# B&R Automation Studio project Genmot_Markalama_
Automation Studio 3.0.90.36 SP18

## Configuration Config1

### Task classes (Cpu.sw)
```
Cyclic#1:
  PowerAx1 <- PowerAx1.prg
  PowerAx2 <- PowerAx2.prg
  RZAxisCont <- RZAxisControl.prg
  RYAxisCont <- RYAxisControl.prg
  RXAxisCont <- RXAxisControl.prg
  RAAxisCont <- RAAxisControl.prg
  RC1AxisCon <- RC1AxisControl.prg
  RC2AxisCon <- RC2AxisControl.prg
  GRXAxisCon <- GRXAxisControl.prg
  GRZAxisCon <- GRZAxisControl.prg
  Master <- Master.prg
Cyclic#2:
  Sender <- LibDVFrame1_ST.Sender.prg
  Receiver <- LibDVFrame1_ST.Receiver.prg
Cyclic#4:
  GRYAxisCon <- GRYAxisControl.prg
DataObjects: Acp10sys
NcDataObjects: acp10etxen <- acp10etxen.dob, gaxis01i <- RYAxisobj.gaxis01i.dob, gaxis01a <- RYAxisobj.gaxis01a.dob, gaxis02i <- RAAxisobj.gaxis02i.dob, gaxis02a <- RAAxisobj.gaxis02a.dob, gaxis03i <- RXAxisobj.gaxis03i.dob, gaxis03a <- RXAxisobj.gaxis03a.dob, gz1_axisi <- RZAxisobj.gz1_axisi.dob, gz1_axisa <- RZAxisobj.gz1_axisa.dob, gc1_axisi <- RC1Axisobj.gc1_axisi.dob, gc2_axisa <- RC1Axisobj.gc2_axisa.dob, gc2_axisi <- RC2Axisobj.gc2_axisi.dob, gc2_axisa1 <- RC2Axisobj.gc2_axisa.dob, powersp1i <- PowerSp1obj.powersp1i.dob, powersp1a <- PowerSp1obj.powersp1a.dob, powersp2i <- PowerSp2obj.powersp2i.dob, powersp2a <- PowerSp2obj.powersp2a.dob, grx_axisi <- GRXAxisobj.grx_axisi.dob, grx_axisa <- GRXAxisobj.grx_axisa.dob, grz_axisi <- GRZAxisobj.grz_axisi.dob, grz_axisa <- GRZAxisobj.grz_axisa.dob, gry_axisi <- GRYAxisobj.gry_axisi.dob, gry_axisa <- GRYAxisobj.gry_axisa.dob
Binaries: AsOPCC, ashwd, arconfig, sysconf, asfw, iomap, Acp10cfg, Acp10map, Visu03, vcctrend, vccline, vcchtml, vcbclass, vccbmp, vcclbox, vccalarm, vcrt, vcshared, vcnet, arialbd, vcdsloc, vcgclass, vcresman, vccstr, vcmgr, vcfile, vcalarm, vccurl, vcpdsw, Visu02, vcpdvnc, vcdsint, vccnum, vccbtn, vcpfar10, vcpkat, vctcal, arial, vccovl, vcctext, vccshape, vcfntttf, vcxml, Visu01, visvc, vccbar
Libraries: acp10_mc, brsystem, Acp10man, sys_lib, NcGlobal, Acp10par, runtime, Acp10sdc, standard, asstring, astime, powerlnk, AsWeigh, AsBrMath, LoopConR, AsBrStr, FileIO, AsEPL, AsARCfg, asieccon, dvframe, ashw, dataobj, visapi
```

### Cpu.per - PLC1/Cpu.per
```iecst
(********************************************************************
 * COPYRIGHT --
 ********************************************************************
 * File: Cpu.per
 * Author: Coder
 * Created: September 22, 2013
 ********************************************************************
 * Declaration of permanent variables
 ********************************************************************)
VAR_CONFIG
	Retain AT %M0;
	Eksen_Hizlari AT %M76;
END_VAR
```

### IoMap.iom - PLC1/IoMap.iom
```iecst
(********************************************************************
 * COPYRIGHT --
 ********************************************************************
 * File: IoMap.iom
 * Author: Coder
 * Created: September 22, 2013
 ********************************************************************
 * IO mapping file
 ********************************************************************)
VAR_CONFIG
	DI.Acil_Stop AT %IX.SL1.IF1.ST1.IF1.ST2.DigitalInput01;
	DI.X_PosLimit AT %IX.SL1.IF1.ST1.IF1.ST2.DigitalInput03;
	DI.X_NegLimit AT %IX.SL1.IF1.ST1.IF1.ST2.DigitalInput04;
	DI.X_RefSensor AT %IX.SL1.IF1.ST1.IF1.ST2.DigitalInput02;
	DI.Y_NegLimit AT %IX.SL1.IF1.ST1.IF1.ST2.DigitalInput06;
	DI.Y_RefSensor AT %IX.SL1.IF1.ST1.IF1.ST2.DigitalInput05;
	DI.Y_PosLimit AT %IX.SL1.IF1.ST1.IF1.ST2.DigitalInput07;
	DI.Lazer_IsBitti AT %IX.SL1.IF1.ST1.IF1.ST2.DigitalInput08;
	DI.GRX_PosLimit AT %IX.SL1.IF1.ST1.IF1.ST3.DigitalInput01;
	DI.GRX_RefSensor AT %IX.SL1.IF1.ST1.IF1.ST2.DigitalInput12;
	DI.GRX_NegLimit AT %IX.SL1.IF1.ST1.IF1.ST2.DigitalInput11;
	DI.GRZ_PosLimit AT %IX.SL1.IF1.ST1.IF1.ST3.DigitalInput04;
	DI.GRZ_NegLimit AT %IX.SL1.IF1.ST1.IF1.ST3.DigitalInput03;
	DI.GRZ_RefSensor AT %IX.SL1.IF1.ST1.IF1.ST3.DigitalInput02;
	DI.GRY_NegLimit AT %IX.SL1.IF1.ST1.IF1.ST3.DigitalInput06;
	DQ.Konveyor_Ileri AT %QX.SL1.IF1.ST1.IF1.ST7.DigitalOutput01;
	DQ.Konveyor_Geri AT %QX.SL1.IF1.ST1.IF1.ST7.DigitalOutput02;
	DQ.Lazer_Start AT %QX.SL1.IF1.ST1.IF1.ST6.DigitalOutput01;
	DQ.Lazer_Stop AT %QX.SL1.IF1.ST1.IF1.ST6.DigitalOutput02;
	DQ.Lazer_Pointer AT %QX.SL1.IF1.ST1.IF1.ST6.DigitalOutput03;
	DQ.Lazer_Hatch AT %QX.SL1.IF1.ST1.IF1.ST6.DigitalOutput04;
	DQ.Lazer_Barcode AT %QX.SL1.IF1.ST1.IF1.ST6.DigitalOutput05;
	DQ.Kripper_Ac AT %QX.SL1.IF1.ST1.IF1.ST6.DigitalOutput07;
	DQ.Kripper_Kapat AT %QX.SL1.IF1.ST1.IF1.ST6.DigitalOutput08;
	DI.LAnahtarKonumu1 AT %IX.SL1.IF1.ST1.IF1.ST4.DigitalInput09;
	DI.LAnahtarKonumu2 AT %IX.SL1.IF1.ST1.IF1.ST4.DigitalInput11;
	DI.LAnahtarKonumu3 AT %IX.SL1.IF1.ST1.IF1.ST4.DigitalInput02;
	DI.LAnahtarKonumu4 AT %IX.SL1.IF1.ST1.IF1.ST4.DigitalInput04;
	DI.L_JoySag AT %IX.SL1.IF1.ST1.IF1.ST4.DigitalInput05;
	DI.L_JoySol AT %IX.SL1.IF1.ST1.IF1.ST4.DigitalInput07;
	DI.L_Input1 AT %IX.SL1.IF1.ST1.IF1.ST4.DigitalInput03;
	DI.RAnahtarKonumu1 AT %IX.SL1.IF1.ST1.IF1.ST5.DigitalInput09;
	DI.RAnahtarKonumu2 AT %IX.SL1.IF1.ST1.IF1.ST5.DigitalInput11;
	DI.RAnahtarKonumu3 AT %IX.SL1.IF1.ST1.IF1.ST5.DigitalInput02;
	DI.RAnahtarKonumu4 AT %IX.SL1.IF1.ST1.IF1.ST5.DigitalInput04;
	DI.R_JoySag AT %IX.SL1.IF1.ST1.IF1.ST5.DigitalInput05;
	DI.R_JoySol AT %IX.SL1.IF1.ST1.IF1.ST5.DigitalInput07;
	DI.R_Input1 AT %IX.SL1.IF1.ST1.IF1.ST5.DigitalInput03;
END_VAR
```

### LazerOpcMap.opcm - PLC1/LazerOpcMap.opcm
```
Map:
  CommunicationPath:
    Pvi (CommunicationTimeout=0, ProcessTimeout=0, RemoutePvi=false, IpAddress=127.0.0.1, PortNumber=20000, Others=)
    Linie LNINA2 (Type=LNINA2, CFG=, Others=)
    Device TCPIP (Type=Tcpip, IF=tcpip, BD=57600, RS=232, PA=1, CNO=0, IT=40, BI=1598, MDA=32, SA=54, CMODE=11, CT=20, MC=15, LOPO=11159, MO='Modem description see Control Panel', TN='+90909090909', MR=INFINITE, RI=60, FF=nw_load.bin, FC=nw_pb_32.br, CB=2, RC=3, TE=3000, TQ=3000, SR=0, RETRY=3, DA=2, TO=100, BA=851968, Others=)
    Station (CN=Station, MODE=SPS, DAIP=, PN=502, Others=)
    Cpu NewTCPIPConnection (CN=, SP=, RT=1000, DA=, DAIP=192.168.137.2, RW=0, REPO=11159, CKDA=1, Others=)
  Tag GC1_MoveAbsolute (Scope=)
    PVI GC1Axis.Command.MoveAbsolute (Path=GC1Axis.Command.MoveAbsolute, Type=Pvar, AccessType=DATA)
      ObjectDescriptor (VT=boolean, VN=1, VL=1, CD=GC1Axis.Command.MoveAbsolute, AT=rw, RF=1000, DV=, WR=true)
      LinkDescriptor (BitNumber=none, LT=raw)
        CastMode (Pg2000=false, Decimal=false, Range=false, Rounding=false, TerminateStrings=false)
  Tag GC1_Position (Scope=)
    PVI GC1Axis.Parameter.Position (Path=GC1Axis.Parameter.Position, Type=Pvar, AccessType=DATA)
      ObjectDescriptor (VT=f32, VN=1, VL=4, CD=GC1Axis.Parameter.Position, AT=rw, RF=1000, DV=, WR=true)
      LinkDescriptor (BitNumber=none, LT=raw)
        CastMode (Pg2000=false, Decimal=false, Range=false, Rounding=false, TerminateStrings=false)
  Tag Markalama_Ok_Delphi (Scope=)
    PVI Parametreler_0.Markalama_Ok_Delphi (Path=Parametreler_0.Markalama_Ok_Delphi, Type=Pvar, AccessType=DATA)
      ObjectDescriptor (VT=boolean, VN=1, VL=1, CD=Parametreler_0.Markalama_Ok_Delphi, AT=rw, RF=1000, DV=, WR=true)
      LinkDescriptor (BitNumber=none, LT=raw)
        CastMode (Pg2000=false, Decimal=false, Range=false, Rounding=false, TerminateStrings=false)
  Tag A_JogVelocity (Scope=)
    PVI Eksen_Hizlari.A_JogVelocity (Path=Eksen_Hizlari.A_JogVelocity, Type=Pvar, AccessType=DATA)
      ObjectDescriptor (VT=f32, VN=1, VL=4, CD=Eksen_Hizlari.A_JogVelocity, AT=rw, RF=1000, DV=, WR=true)
      LinkDescriptor (BitNumber=none, LT=raw)
        CastMode (Pg2000=false, Decimal=false, Range=false, Rounding=false, TerminateStrings=false)
  Tag A_PosVelocity (Scope=)
    PVI Eksen_Hizlari.A_PosVelocity (Path=Eksen_Hizlari.A_PosVelocity, Type=Pvar, AccessType=DATA)
      ObjectDescriptor (VT=f32, VN=1, VL=4, CD=Eksen_Hizlari.A_PosVelocity, AT=rw, RF=1000, DV=, WR=true)
      LinkDescriptor (BitNumber=none, LT=raw)
        CastMode (Pg2000=false, Decimal=false, Range=false, Rounding=false, TerminateStrings=false)
  Tag GC1_JogVelocity (Scope=)
    PVI Eksen_Hizlari.GC1_JogVelocity (Path=Eksen_Hizlari.GC1_JogVelocity, Type=Pvar, AccessType=DATA)
      ObjectDescriptor (VT=f32, VN=1, VL=4, CD=Eksen_Hizlari.GC1_JogVelocity, AT=rw, RF=1000, DV=, WR=true)
      LinkDescriptor (BitNumber=none, LT=raw)
        CastMode (Pg2000=false, Decimal=false, Range=false, Rounding=false, TerminateStrings=false)
  Tag GC1_PosVelocity (Scope=)
    PVI Eksen_Hizlari.GC1_PosVelocity (Path=Eksen_Hizlari.GC1_PosVelocity, Type=Pvar, AccessType=DATA)
      ObjectDescriptor (VT=f32, VN=1, VL=4, CD=Eksen_Hizlari.GC1_PosVelocity, AT=rw, RF=1000, DV=, WR=true)
      LinkDescriptor (BitNumber=none, LT=raw)
        CastMode (Pg2000=false, Decimal=false, Range=false, Rounding=false, TerminateStrings=false)
  Tag GRX_JogVelocity (Scope=)
    PVI Eksen_Hizlari.GRX_JogVelocity (Path=Eksen_Hizlari.GRX_JogVelocity, Type=Pvar, AccessType=DATA)
      ObjectDescriptor (VT=f32, VN=1, VL=4, CD=Eksen_Hizlari.GRX_JogVelocity, AT=rw, RF=1000, DV=, WR=true)
      LinkDescriptor (BitNumber=none, LT=raw)
        CastMode (Pg2000=false, Decimal=false, Range=false, Rounding=false, TerminateStrings=false)
  Tag GRX_PosVelocity (Scope=)
    PVI Eksen_Hizlari.GRX_PosVelocity (Path=Eksen_Hizlari.GRX_PosVelocity, Type=Pvar, AccessType=DATA)
      ObjectDescriptor (VT=f32, VN=1, VL=4, CD=Eksen_Hizlari.GRX_PosVelocity, AT=rw, RF=1000, DV=, WR=true)
      LinkDescriptor (BitNumber=none, LT=raw)
        CastMode (Pg2000=false, Decimal=false, Range=false, Rounding=false, TerminateStrings=false)
  Tag GRY_JogVelocity (Scope=)
    PVI Eksen_Hizlari.GRY_JogVelocity (Path=Eksen_Hizlari.GRY_JogVelocity, Type=Pvar, AccessType=DATA)
      ObjectDescriptor (VT=f32, VN=1, VL=4, CD=Eksen_Hizlari.GRY_JogVelocity, AT=rw, RF=1000, DV=, WR=true)
      LinkDescriptor (BitNumber=none, LT=raw)
        CastMode (Pg2000=false, Decimal=false, Range=false, Rounding=false, TerminateStrings=false)
  Tag GRY_PosVelocity (Scope=)
    PVI Eksen_Hizlari.GRY_PosVelocity (Path=Eksen_Hizlari.GRY_PosVelocity, Type=Pvar, AccessType=DATA)
      ObjectDescriptor (VT=f32, VN=1, VL=4, CD=Eksen_Hizlari.GRY_PosVelocity, AT=rw, RF=1000, DV=, WR=true)
      LinkDescriptor (BitNumber=none, LT=raw)
        CastMode (Pg2000=false, Decimal=false, Range=false, Rounding=false, TerminateStrings=false)
  Tag GRZ_JogVelocity (Scope=)
    PVI Eksen_Hizlari.GRZ_JogVelocity (Path=Eksen_Hizlari.GRZ_JogVelocity, Type=Pvar, AccessType=DATA)
      ObjectDescriptor (VT=f32, VN=1, VL=4, CD=Eksen_Hizlari.GRZ_JogVelocity, AT=rw, RF=1000, DV=, WR=true)
      LinkDescriptor (BitNumber=none, LT=raw)
        CastMode (Pg2000=false, Decimal=false, Range=false, Rounding=false, TerminateStrings=false)
  Tag GRZ_PosVelocity (Scope=)
    PVI Eksen_Hizlari.GRZ_PosVelocity (Path=Eksen_Hizlari.GRZ_PosVelocity, Type=Pvar, AccessType=DATA)
      ObjectDescriptor (VT=f32, VN=1, VL=4, CD=Eksen_Hizlari.GRZ_PosVelocity, AT=rw, RF=1000, DV=, WR=true)
      LinkDescriptor (BitNumber=none, LT=raw)
        CastMode (Pg2000=false, Decimal=false, Range=false, Rounding=false, TerminateStrings=false)
  Tag X_JogVelocity (Scope=)
    PVI Eksen_Hizlari.X_JogVelocity (Path=Eksen_Hizlari.X_JogVelocity, Type=Pvar, AccessType=DATA)
      ObjectDescriptor (VT=f32, VN=1, VL=4, CD=Eksen_Hizlari.X_JogVelocity, AT=rw, RF=1000, DV=, WR=true)
      LinkDescriptor (BitNumber=none, LT=raw)
        CastMode (Pg2000=false, Decimal=false, Range=false, Rounding=false, TerminateStrings=false)
  Tag X_PosVelocity (Scope=)
    PVI Eksen_Hizlari.X_PosVelocity (Path=Eksen_Hizlari.X_PosVelocity, Type=Pvar, AccessType=DATA)
      ObjectDescriptor (VT=f32, VN=1, VL=4, CD=Eksen_Hizlari.X_PosVelocity, AT=rw, RF=1000, DV=, WR=true)
      LinkDescriptor (BitNumber=none, LT=raw)
        CastMode (Pg2000=false, Decimal=false, Range=false, Rounding=false, TerminateStrings=false)
  Tag Y_JogVelocity (Scope=)
    PVI Eksen_Hizlari.Y_JogVelocity (Path=Eksen_Hizlari.Y_JogVelocity, Type=Pvar, AccessType=DATA)
      ObjectDescriptor (VT=f32, VN=1, VL=4, CD=Eksen_Hizlari.Y_JogVelocity, AT=rw, RF=1000, DV=, WR=true)
      LinkDescriptor (BitNumber=none, LT=raw)
        CastMode (Pg2000=false, Decimal=false, Range=false, Rounding=false, TerminateStrings=false)
  Tag Y_PosVelocity (Scope=)
    PVI Eksen_Hizlari.Y_PosVelocity (Path=Eksen_Hizlari.Y_PosVelocity, Type=Pvar, AccessType=DATA)
      ObjectDescriptor (VT=f32, VN=1, VL=4, CD=Eksen_Hizlari.Y_PosVelocity, AT=rw, RF=1000, DV=, WR=true)
      LinkDescriptor (BitNumber=none, LT=raw)
        CastMode (Pg2000=false, Decimal=false, Range=false, Rounding=false, TerminateStrings=false)
  Tag Z_JogVelocity (Scope=)
    PVI Eksen_Hizlari.Z_JogVelocity (Path=Eksen_Hizlari.Z_JogVelocity, Type=Pvar, AccessType=DATA)
      ObjectDescriptor (VT=f32, VN=1, VL=4, CD=Eksen_Hizlari.Z_JogVelocity, AT=rw, RF=1000, DV=, WR=true)
      LinkDescriptor (BitNumber=none, LT=raw)
        CastMode (Pg2000=false, Decimal=false, Range=false, Rounding=false, TerminateStrings=false)
  Tag Z_PosVelocity (Scope=)
    PVI Eksen_Hizlari.Z_PosVelocity (Path=Eksen_Hizlari.Z_PosVelocity, Type=Pvar, AccessType=DATA)
      ObjectDescriptor (VT=f32, VN=1, VL=4, CD=Eksen_Hizlari.Z_PosVelocity, AT=rw, RF=1000, DV=, WR=true)
      LinkDescriptor (BitNumber=none, LT=raw)
        CastMode (Pg2000=false, Decimal=false, Range=false, Rounding=false, TerminateStrings=false)
  Tag GRY_Actual_Pos_mm (Scope=)
    PVI Actual_Pos.GRY_Actual_Pos (Path=Actual_Pos.GRY_Actual_Pos, Type=Pvar, AccessType=DATA)
      ObjectDescriptor (VT=f32, VN=1, VL=4, CD=Actual_Pos.GRY_Actual_Pos, AT=rw, RF=1000, DV=, WR=true)
      LinkDescriptor (BitNumber=none, LT=raw)
        CastMode (Pg2000=false, Decimal=false, Range=false, Rounding=false, TerminateStrings=false)
  Tag GRY_HedefPozisyon (Scope=)
    PVI Retain.GRY_KrankAlma_Konumu (Path=Retain.GRY_KrankAlma_Konumu, Type=Pvar, AccessType=DATA)
      ObjectDescriptor (VT=f32, VN=1, VL=4, CD=Retain.GRY_KrankAlma_Konumu, AT=rw, RF=1000, DV=, WR=true)
      LinkDescriptor (BitNumber=none, LT=raw)
        CastMode (Pg2000=false, Decimal=false, Range=false, Rounding=false, TerminateStrings=false)
  Tag GRX_HedefPozisyon (Scope=)
    PVI Parametreler_0.GRX_Position (Path=Parametreler_0.GRX_Position, Type=Pvar, AccessType=DATA)
      ObjectDescriptor (VT=f32, VN=1, VL=4, CD=Parametreler_0.GRX_Position, AT=rw, RF=1000, DV=, WR=true)
      LinkDescriptor (BitNumber=none, LT=raw)
        CastMode (Pg2000=false, Decimal=false, Range=false, Rounding=false, TerminateStrings=false)
  Tag GRZ_HedefPozisyon (Scope=)
    PVI Parametreler_0.GRZ_Position (Path=Parametreler_0.GRZ_Position, Type=Pvar, AccessType=DATA)
      ObjectDescriptor (VT=f32, VN=1, VL=4, CD=Parametreler_0.GRZ_Position, AT=rw, RF=1000, DV=, WR=true)
      LinkDescriptor (BitNumber=none, LT=raw)
        CastMode (Pg2000=false, Decimal=false, Range=false, Rounding=false, TerminateStrings=false)
  Tag GC1_ErrorID (Scope=)
    PVI GC1Axis.Status.ErrorID (Path=GC1Axis.Status.ErrorID, Type=Pvar, AccessType=DATA)
      ObjectDescriptor (VT=u16, VN=1, VL=2, CD=GC1Axis.Status.ErrorID, AT=rw, RF=1000, DV=, WR=true)
      LinkDescriptor (BitNumber=none, LT=raw)
        CastMode (Pg2000=false, Decimal=false, Range=false, Rounding=false, TerminateStrings=false)
  Tag GC2_ErrorID (Scope=)
    PVI GC2Axis.Status.ErrorID (Path=GC2Axis.Status.ErrorID, Type=Pvar, AccessType=DATA)
      ObjectDescriptor (VT=u16, VN=1, VL=2, CD=GC2Axis.Status.ErrorID, AT=rw, RF=1000, DV=, WR=true)
      LinkDescriptor (BitNumber=none, LT=raw)
        CastMode (Pg2000=false, Decimal=false, Range=false, Rounding=false, TerminateStrings=false)
  Tag GRX_ErrorID (Scope=)
    PVI GRXAxis.Status.ErrorID (Path=GRXAxis.Status.ErrorID, Type=Pvar, AccessType=DATA)
      ObjectDescriptor (VT=u16, VN=1, VL=2, CD=GRXAxis.Status.ErrorID, AT=rw, RF=1000, DV=, WR=true)
      LinkDescriptor (BitNumber=none, LT=raw)
        CastMode (Pg2000=false, Decimal=false, Range=false, Rounding=false, TerminateStrings=false)
  Tag GRY_ErrorID (Scope=)
    PVI GRYAxis.Status.ErrorID (Path=GRYAxis.Status.ErrorID, Type=Pvar, AccessType=DATA)
      ObjectDescriptor (VT=u16, VN=1, VL=2, CD=GRYAxis.Status.ErrorID, AT=rw, RF=1000, DV=, WR=true)
      LinkDescriptor (BitNumber=none, LT=raw)
        CastMode (Pg2000=false, Decimal=false, Range=false, Rounding=false, TerminateStrings=false)
  Tag GRZ_ErrorID (Scope=)
    PVI GRZAxis.Status.ErrorID (Path=GRZAxis.Status.ErrorID, Type=Pvar, AccessType=DATA)
      ObjectDescriptor (VT=u16, VN=1, VL=2, CD=GRZAxis.Status.ErrorID, AT=rw, RF=1000, DV=, WR=true)
      LinkDescriptor (BitNumber=none, LT=raw)
        CastMode (Pg2000=false, Decimal=false, Range=false, Rounding=false, TerminateStrings=false)
  Tag Kripper_Ac (Scope=)
    PVI Parametreler_0.Kripper_Ac (Path=Parametreler_0.Kripper_Ac, Type=Pvar, AccessType=DATA)
      ObjectDescriptor (VT=boolean, VN=1, VL=1, CD=Parametreler_0.Kripper_Ac, AT=rw, RF=1000, DV=, WR=true)
      LinkDescriptor (BitNumber=none, LT=raw)
        CastMode (Pg2000=false, Decimal=false, Range=false, Rounding=false, TerminateStrings=false)
  Tag Kripper_Kapat (Scope=)
    PVI Parametreler_0.Kripper_Kapat (Path=Parametreler_0.Kripper_Kapat, Type=Pvar, AccessType=DATA)
      ObjectDescriptor (VT=boolean, VN=1, VL=1, CD=Parametreler_0.Kripper_Kapat, AT=rw, RF=1000, DV=, WR=true)
      LinkDescriptor (BitNumber=none, LT=raw)
        CastMode (Pg2000=false, Decimal=false, Range=false, Rounding=false, TerminateStrings=false)
  Tag RA_ErrorID (Scope=)
    PVI GX1Axis.Status.ErrorID (Path=GX1Axis.Status.ErrorID, Type=Pvar, AccessType=DATA)
      ObjectDescriptor (VT=u16, VN=1, VL=2, CD=GX1Axis.Status.ErrorID, AT=rw, RF=1000, DV=, WR=true)
      LinkDescriptor (BitNumber=none, LT=raw)
        CastMode (Pg2000=false, Decimal=false, Range=false, Rounding=false, TerminateStrings=false)
  Tag RX_ErrorID (Scope=)
    PVI GX2Axis.Status.ErrorID (Path=GX2Axis.Status.ErrorID, Type=Pvar, AccessType=DATA)
      ObjectDescriptor (VT=u16, VN=1, VL=2, CD=GX2Axis.Status.ErrorID, AT=rw, RF=1000, DV=, WR=true)
      LinkDescriptor (BitNumber=none, LT=raw)
        CastMode (Pg2000=false, Decimal=false, Range=false, Rounding=false, TerminateStrings=false)
  Tag RY_ErrorID (Scope=)
    PVI GX3Axis.Status.ErrorID (Path=GX3Axis.Status.ErrorID, Type=Pvar, AccessType=DATA)
      ObjectDescriptor (VT=u16, VN=1, VL=2, CD=GX3Axis.Status.ErrorID, AT=rw, RF=1000, DV=, WR=true)
      LinkDescriptor (BitNumber=none, LT=raw)
        CastMode (Pg2000=false, Decimal=false, Range=false, Rounding=false, TerminateStrings=false)
  Tag RZ_ErrorID (Scope=)
    PVI GZ1Axis.Status.ErrorID (Path=GZ1Axis.Status.ErrorID, Type=Pvar, AccessType=DATA)
      ObjectDescriptor (VT=u16, VN=1, VL=2, CD=GZ1Axis.Status.ErrorID, AT=rw, RF=1000, DV=, WR=true)
      LinkDescriptor (BitNumber=none, LT=raw)
        CastMode (Pg2000=false, Decimal=false, Range=false, Rounding=false, TerminateStrings=false)
  Tag Markalama_Git (Scope=)
    PVI Parametreler_0.Markalamaya_Git (Path=Parametreler_0.Markalamaya_Git, Type=Pvar, AccessType=DATA)
      ObjectDescriptor (VT=boolean, VN=1, VL=1, CD=Parametreler_0.Markalamaya_Git, AT=rw, RF=1000, DV=, WR=true)
      LinkDescriptor (BitNumber=none, LT=raw)
        CastMode (Pg2000=false, Decimal=false, Range=false, Rounding=false, TerminateStrings=false)
  Tag Markalama_Start (Scope=)
    PVI Parametreler_0.Markalama_Start (Path=Parametreler_0.Markalama_Start, Type=Pvar, AccessType=DATA)
      ObjectDescriptor (VT=boolean, VN=1, VL=1, CD=Parametreler_0.Markalama_Start, AT=rw, RF=1000, DV=, WR=true)
      LinkDescriptor (BitNumber=none, LT=raw)
        CastMode (Pg2000=false, Decimal=false, Range=false, Rounding=false, TerminateStrings=false)
  Tag Markalama_Ok (Scope=)
    PVI Parametreler_0.Markalama_Ok (Path=Parametreler_0.Markalama_Ok, Type=Pvar, AccessType=DATA)
      ObjectDescriptor (VT=boolean, VN=1, VL=1, CD=Parametreler_0.Markalama_Ok, AT=rw, RF=1000, DV=, WR=true)
      LinkDescriptor (BitNumber=none, LT=raw)
        CastMode (Pg2000=false, Decimal=false, Range=false, Rounding=false, TerminateStrings=false)
  Tag GRY_JogPos (Scope=)
    PVI Parametreler_0.GRY_JogPos (Path=Parametreler_0.GRY_JogPos, Type=Pvar, AccessType=DATA)
      ObjectDescriptor (VT=boolean, VN=1, VL=1, CD=Parametreler_0.GRY_JogPos, AT=rw, RF=1000, DV=, WR=true)
      LinkDescriptor (BitNumber=none, LT=raw)
        CastMode (Pg2000=false, Decimal=false, Range=false, Rounding=false, TerminateStrings=false)
  Tag GRY_JogNeg (Scope=)
    PVI Parametreler_0.GRY_JogNeg (Path=Parametreler_0.GRY_JogNeg, Type=Pvar, AccessType=DATA)
      ObjectDescriptor (VT=boolean, VN=1, VL=1, CD=Parametreler_0.GRY_JogNeg, AT=rw, RF=1000, DV=, WR=true)
      LinkDescriptor (BitNumber=none, LT=raw)
        CastMode (Pg2000=false, Decimal=false, Range=false, Rounding=false, TerminateStrings=false)
  Tag GRY_HomeStart (Scope=)
    PVI Parametreler_0.GRY_HomeStart (Path=Parametreler_0.GRY_HomeStart, Type=Pvar, AccessType=DATA)
      ObjectDescriptor (VT=boolean, VN=1, VL=1, CD=Parametreler_0.GRY_HomeStart, AT=rw, RF=1000, DV=, WR=true)
      LinkDescriptor (BitNumber=none, LT=raw)
        CastMode (Pg2000=false, Decimal=false, Range=false, Rounding=false, TerminateStrings=false)
  Tag GRY_HomeOk (Scope=)
    PVI Parametreler_0.GRY_HomeOk (Path=Parametreler_0.GRY_HomeOk, Type=Pvar, AccessType=DATA)
      ObjectDescriptor (VT=boolean, VN=1, VL=1, CD=Parametreler_0.GRY_HomeOk, AT=rw, RF=1000, DV=, WR=true)
      LinkDescriptor (BitNumber=none, LT=raw)
        CastMode (Pg2000=false, Decimal=false, Range=false, Rounding=false, TerminateStrings=false)
  Tag Konveyor_Geri_Buton (Scope=)
    PVI Parametreler_0.Konveyor_Geri_Buton (Path=Parametreler_0.Konveyor_Geri_Buton, Type=Pvar, AccessType=DATA)
      ObjectDescriptor (VT=boolean, VN=1, VL=1, CD=Parametreler_0.Konveyor_Geri_Buton, AT=rw, RF=1000, DV=, WR=true)
      LinkDescriptor (BitNumber=none, LT=raw)
        CastMode (Pg2000=false, Decimal=false, Range=false, Rounding=false, TerminateStrings=false)
  Tag Konveyor_Ileri_Buton (Scope=)
    PVI Parametreler_0.Konveyor_Ileri_Buton (Path=Parametreler_0.Konveyor_Ileri_Buton, Type=Pvar, AccessType=DATA)
      ObjectDescriptor (VT=boolean, VN=1, VL=1, CD=Parametreler_0.Konveyor_Ileri_Buton, AT=rw, RF=1000, DV=, WR=true)
      LinkDescriptor (BitNumber=none, LT=raw)
        CastMode (Pg2000=false, Decimal=false, Range=false, Rounding=false, TerminateStrings=false)
  Tag Dikey_Sira_Araligi (Scope=)
    PVI Retain.Dikey_Sira_Araligi (Path=Retain.Dikey_Sira_Araligi, Type=Pvar, AccessType=DATA)
      ObjectDescriptor (VT=f32, VN=1, VL=4, CD=Retain.Dikey_Sira_Araligi, AT=rw, RF=1000, DV=, WR=true)
      LinkDescriptor (BitNumber=none, LT=raw)
        CastMode (Pg2000=false, Decimal=false, Range=false, Rounding=false, TerminateStrings=false)
  Tag Dikey_Sira_Miktari (Scope=)
    PVI Retain.Dikey_Sira_Miktari (Path=Retain.Dikey_Sira_Miktari, Type=Pvar, AccessType=DATA)
      ObjectDescriptor (VT=u8, VN=1, VL=1, CD=Retain.Dikey_Sira_Miktari, AT=rw, RF=1000, DV=, WR=true)
      LinkDescriptor (BitNumber=none, LT=raw)
        CastMode (Pg2000=false, Decimal=false, Range=false, Rounding=false, TerminateStrings=false)
  Tag Yatay_Sira_Araligi (Scope=)
    PVI Retain.Yatay_Sira_Araligi (Path=Retain.Yatay_Sira_Araligi, Type=Pvar, AccessType=DATA)
      ObjectDescriptor (VT=f32, VN=1, VL=4, CD=Retain.Yatay_Sira_Araligi, AT=rw, RF=1000, DV=, WR=true)
      LinkDescriptor (BitNumber=none, LT=raw)
        CastMode (Pg2000=false, Decimal=false, Range=false, Rounding=false, TerminateStrings=false)
  Tag Yatay_Sira_Miktari (Scope=)
    PVI Retain.Yatay_Sira_Miktari (Path=Retain.Yatay_Sira_Miktari, Type=Pvar, AccessType=DATA)
      ObjectDescriptor (VT=u8, VN=1, VL=1, CD=Retain.Yatay_Sira_Miktari, AT=rw, RF=1000, DV=, WR=true)
      LinkDescriptor (BitNumber=none, LT=raw)
        CastMode (Pg2000=false, Decimal=false, Range=false, Rounding=false, TerminateStrings=false)
  Tag GRX_KrankAlma_Konumu_2 (Scope=)
    PVI Retain.GRX_KrankAlma_Konumu_2 (Path=Retain.GRX_KrankAlma_Konumu_2, Type=Pvar, AccessType=DATA)
      ObjectDescriptor (VT=f32, VN=1, VL=4, CD=Retain.GRX_KrankAlma_Konumu_2, AT=rw, RF=1000, DV=, WR=true)
      LinkDescriptor (BitNumber=none, LT=raw)
        CastMode (Pg2000=false, Decimal=false, Range=false, Rounding=false, TerminateStrings=false)
  Tag GRX_KrankKoyma_Konumu_2 (Scope=)
    PVI Retain.GRX_KrankKoyma_Konumu_2 (Path=Retain.GRX_KrankKoyma_Konumu_2, Type=Pvar, AccessType=DATA)
      ObjectDescriptor (VT=f32, VN=1, VL=4, CD=Retain.GRX_KrankKoyma_Konumu_2, AT=rw, RF=1000, DV=, WR=true)
      LinkDescriptor (BitNumber=none, LT=raw)
        CastMode (Pg2000=false, Decimal=false, Range=false, Rounding=false, TerminateStrings=false)
  Tag GRZ_KrankAlma_Konumu_2 (Scope=)
    PVI Retain.GRZ_KrankAlma_Konumu_2 (Path=Retain.GRZ_KrankAlma_Konumu_2, Type=Pvar, AccessType=DATA)
      ObjectDescriptor (VT=f32, VN=1, VL=4, CD=Retain.GRZ_KrankAlma_Konumu_2, AT=rw, RF=1000, DV=, WR=true)
      LinkDescriptor (BitNumber=none, LT=raw)
        CastMode (Pg2000=false, Decimal=false, Range=false, Rounding=false, TerminateStrings=false)
  Tag GRZ_KrankKoyma_Konumu_2 (Scope=)
    PVI Retain.GRZ_KrankKoyma_Konumu_2 (Path=Retain.GRZ_KrankKoyma_Konumu_2, Type=Pvar, AccessType=DATA)
      ObjectDescriptor (VT=f32, VN=1, VL=4, CD=Retain.GRZ_KrankKoyma_Konumu_2, AT=rw, RF=1000, DV=, WR=true)
      LinkDescriptor (BitNumber=none, LT=raw)
        CastMode (Pg2000=false, Decimal=false, Range=false, Rounding=false, TerminateStrings=false)
  Tag Krank_Koy (Scope=)
    PVI Parametreler_0.Krank_Koy (Path=Parametreler_0.Krank_Koy, Type=Pvar, AccessType=DATA)
      ObjectDescriptor (VT=boolean, VN=1, VL=1, CD=Parametreler_0.Krank_Koy, AT=rw, RF=1000, DV=, WR=true)
      LinkDescriptor (BitNumber=none, LT=raw)
        CastMode (Pg2000=false, Decimal=false, Range=false, Rounding=false, TerminateStrings=false)
  Tag GRX_KrankAlmaKonumu (Scope=)
    PVI Retain.GRX_KrankAlmaKonumu (Path=Retain.GRX_KrankAlmaKonumu, Type=Pvar, AccessType=DATA)
      ObjectDescriptor (VT=f32, VN=1, VL=4, CD=Retain.GRX_KrankAlmaKonumu, AT=rw, RF=1000, DV=, WR=true)
      LinkDescriptor (BitNumber=none, LT=raw)
        CastMode (Pg2000=false, Decimal=false, Range=false, Rounding=false, TerminateStrings=false)
  Tag GRX_KrankKoymaKonumu (Scope=)
    PVI Retain.GRX_KrankKoymaKonumu (Path=Retain.GRX_KrankKoymaKonumu, Type=Pvar, AccessType=DATA)
      ObjectDescriptor (VT=f32, VN=1, VL=4, CD=Retain.GRX_KrankKoymaKonumu, AT=rw, RF=1000, DV=, WR=true)
      LinkDescriptor (BitNumber=none, LT=raw)
        CastMode (Pg2000=false, Decimal=false, Range=false, Rounding=false, TerminateStrings=false)
  Tag GRZ_KrankAlmaKonumu (Scope=)
    PVI Retain.GRZ_KrankAlmaKonumu (Path=Retain.GRZ_KrankAlmaKonumu, Type=Pvar, AccessType=DATA)
      ObjectDescriptor (VT=f32, VN=1, VL=4, CD=Retain.GRZ_KrankAlmaKonumu, AT=rw, RF=1000, DV=, WR=true)
      LinkDescriptor (BitNumber=none, LT=raw)
        CastMode (Pg2000=false, Decimal=false, Range=false, Rounding=false, TerminateStrings=false)
  Tag GRZ_KrankKoymaKonumu (Scope=)
    PVI Retain.GRZ_KrankKoymaKonumu (Path=Retain.GRZ_KrankKoymaKonumu, Type=Pvar, AccessType=DATA)
      ObjectDescriptor (VT=f32, VN=1, VL=4, CD=Retain.GRZ_KrankKoymaKonumu, AT=rw, RF=1000, DV=, WR=true)
      LinkDescriptor (BitNumber=none, LT=raw)
        CastMode (Pg2000=false, Decimal=false, Range=false, Rounding=false, TerminateStrings=false)
  Tag A_Act_Pos_mm (Scope=)
    PVI Actual_Pos.RA_Actual_Pos (Path=Actual_Pos.RA_Actual_Pos, Type=Pvar, AccessType=DATA)
      ObjectDescriptor (VT=f32, VN=1, VL=4, CD=Actual_Pos.RA_Actual_Pos, AT=rw, RF=1000, DV=, WR=true)
      LinkDescriptor (BitNumber=none, LT=raw)
        CastMode (Pg2000=false, Decimal=false, Range=false, Rounding=false, TerminateStrings=false)
  Tag A_JogNeg (Scope=)
    PVI Parametreler_0.A_JogNeg (Path=Parametreler_0.A_JogNeg, Type=Pvar, AccessType=DATA)
      ObjectDescriptor (VT=boolean, VN=1, VL=1, CD=Parametreler_0.A_JogNeg, AT=rw, RF=1000, DV=, WR=true)
      LinkDescriptor (BitNumber=none, LT=raw)
        CastMode (Pg2000=false, Decimal=false, Range=false, Rounding=false, TerminateStrings=false)
  Tag A_JogPos (Scope=)
    PVI Parametreler_0.A_JogPos (Path=Parametreler_0.A_JogPos, Type=Pvar, AccessType=DATA)
      ObjectDescriptor (VT=boolean, VN=1, VL=1, CD=Parametreler_0.A_JogPos, AT=rw, RF=1000, DV=, WR=true)
      LinkDescriptor (BitNumber=none, LT=raw)
        CastMode (Pg2000=false, Decimal=false, Range=false, Rounding=false, TerminateStrings=false)
  Tag A_Markalama_Konumu (Scope=)
    PVI Retain.RA_MarkalamaKonumu (Path=Retain.RA_MarkalamaKonumu, Type=Pvar, AccessType=DATA)
      ObjectDescriptor (VT=f32, VN=1, VL=4, CD=Retain.RA_MarkalamaKonumu, AT=rw, RF=1000, DV=, WR=true)
      LinkDescriptor (BitNumber=none, LT=raw)
        CastMode (Pg2000=false, Decimal=false, Range=false, Rounding=false, TerminateStrings=false)
  Tag A_Start_Home (Scope=)
    PVI Parametreler_0.A_HomeStart (Path=Parametreler_0.A_HomeStart, Type=Pvar, AccessType=DATA)
      ObjectDescriptor (VT=boolean, VN=1, VL=1, CD=Parametreler_0.A_HomeStart, AT=rw, RF=1000, DV=, WR=true)
      LinkDescriptor (BitNumber=none, LT=raw)
        CastMode (Pg2000=false, Decimal=false, Range=false, Rounding=false, TerminateStrings=false)
  Tag Alarm_Reset (Scope=)
    PVI Parametreler_0.Alarm_Reset (Path=Parametreler_0.Alarm_Reset, Type=Pvar, AccessType=DATA)
      ObjectDescriptor (VT=boolean, VN=1, VL=1, CD=Parametreler_0.Alarm_Reset, AT=rw, RF=1000, DV=, WR=true)
      LinkDescriptor (BitNumber=none, LT=raw)
        CastMode (Pg2000=false, Decimal=false, Range=false, Rounding=false, TerminateStrings=false)
  Tag GC1_Act_Pos_mm (Scope=)
    PVI Actual_Pos.GC1_Actual_Pos (Path=Actual_Pos.GC1_Actual_Pos, Type=Pvar, AccessType=DATA)
      ObjectDescriptor (VT=f32, VN=1, VL=4, CD=Actual_Pos.GC1_Actual_Pos, AT=rw, RF=1000, DV=, WR=true)
      LinkDescriptor (BitNumber=none, LT=raw)
        CastMode (Pg2000=false, Decimal=false, Range=false, Rounding=false, TerminateStrings=false)
  Tag GC1_HomeOk (Scope=)
    PVI Parametreler_0.GC1_HomeOk (Path=Parametreler_0.GC1_HomeOk, Type=Pvar, AccessType=DATA)
      ObjectDescriptor (VT=boolean, VN=1, VL=1, CD=Parametreler_0.GC1_HomeOk, AT=rw, RF=1000, DV=, WR=true)
      LinkDescriptor (BitNumber=none, LT=raw)
        CastMode (Pg2000=false, Decimal=false, Range=false, Rounding=false, TerminateStrings=false)
  Tag GC1_JogNeg (Scope=)
    PVI Parametreler_0.GC1_JogNeg (Path=Parametreler_0.GC1_JogNeg, Type=Pvar, AccessType=DATA)
      ObjectDescriptor (VT=boolean, VN=1, VL=1, CD=Parametreler_0.GC1_JogNeg, AT=rw, RF=1000, DV=, WR=true)
      LinkDescriptor (BitNumber=none, LT=raw)
        CastMode (Pg2000=false, Decimal=false, Range=false, Rounding=false, TerminateStrings=false)
  Tag GC1_JogPos (Scope=)
    PVI Parametreler_0.GC1_JogPos (Path=Parametreler_0.GC1_JogPos, Type=Pvar, AccessType=DATA)
      ObjectDescriptor (VT=boolean, VN=1, VL=1, CD=Parametreler_0.GC1_JogPos, AT=rw, RF=1000, DV=, WR=true)
      LinkDescriptor (BitNumber=none, LT=raw)
        CastMode (Pg2000=false, Decimal=false, Range=false, Rounding=false, TerminateStrings=false)
  Tag GC1_Start_Home (Scope=)
    PVI Parametreler_0.GC1_HomeStart (Path=Parametreler_0.GC1_HomeStart, Type=Pvar, AccessType=DATA)
      ObjectDescriptor (VT=boolean, VN=1, VL=1, CD=Parametreler_0.GC1_HomeStart, AT=rw, RF=1000, DV=, WR=true)
      LinkDescriptor (BitNumber=none, LT=raw)
        CastMode (Pg2000=false, Decimal=false, Range=false, Rounding=false, TerminateStrings=false)
  Tag GC2_Act_Pos_mm (Scope=)
    PVI Actual_Pos.GC2_Actual_Pos (Path=Actual_Pos.GC2_Actual_Pos, Type=Pvar, AccessType=DATA)
      ObjectDescriptor (VT=f32, VN=1, VL=4, CD=Actual_Pos.GC2_Actual_Pos, AT=rw, RF=1000, DV=, WR=true)
      LinkDescriptor (BitNumber=none, LT=raw)
        CastMode (Pg2000=false, Decimal=false, Range=false, Rounding=false, TerminateStrings=false)
  Tag GC2_HomeOk (Scope=)
    PVI Parametreler_0.GC2_HomeOk (Path=Parametreler_0.GC2_HomeOk, Type=Pvar, AccessType=DATA)
      ObjectDescriptor (VT=boolean, VN=1, VL=1, CD=Parametreler_0.GC2_HomeOk, AT=rw, RF=1000, DV=, WR=true)
      LinkDescriptor (BitNumber=none, LT=raw)
        CastMode (Pg2000=false, Decimal=false, Range=false, Rounding=false, TerminateStrings=false)
  Tag GC2_JogNeg (Scope=)
    PVI Parametreler_0.GC2_JogNeg (Path=Parametreler_0.GC2_JogNeg, Type=Pvar, AccessType=DATA)
      ObjectDescriptor (VT=boolean, VN=1, VL=1, CD=Parametreler_0.GC2_JogNeg, AT=rw, RF=1000, DV=, WR=true)
      LinkDescriptor (BitNumber=none, LT=raw)
        CastMode (Pg2000=false, Decimal=false, Range=false, Rounding=false, TerminateStrings=false)
  Tag GC2_JogPos (Scope=)
    PVI Parametreler_0.GC2_JogPos (Path=Parametreler_0.GC2_JogPos, Type=Pvar, AccessType=DATA)
      ObjectDescriptor (VT=boolean, VN=1, VL=1, CD=Parametreler_0.GC2_JogPos, AT=rw, RF=1000, DV=, WR=true)
      LinkDescriptor (BitNumber=none, LT=raw)
        CastMode (Pg2000=false, Decimal=false, Range=false, Rounding=false, TerminateStrings=false)
  Tag GC2_Start_Home (Scope=)
    PVI Parametreler_0.GC2_HomeStart (Path=Parametreler_0.GC2_HomeStart, Type=Pvar, AccessType=DATA)
      ObjectDescriptor (VT=boolean, VN=1, VL=1, CD=Parametreler_0.GC2_HomeStart, AT=rw, RF=1000, DV=, WR=true)
      LinkDescriptor (BitNumber=none, LT=raw)
        CastMode (Pg2000=false, Decimal=false, Range=false, Rounding=false, TerminateStrings=false)
  Tag GRX_Act_Pos_mm (Scope=)
    PVI Actual_Pos.GRX_Actual_Pos (Path=Actual_Pos.GRX_Actual_Pos, Type=Pvar, AccessType=DATA)
      ObjectDescriptor (VT=f32, VN=1, VL=4, CD=Actual_Pos.GRX_Actual_Pos, AT=rw, RF=1000, DV=, WR=true)
      LinkDescriptor (BitNumber=none, LT=raw)
        CastMode (Pg2000=false, Decimal=false, Range=false, Rounding=false, TerminateStrings=false)
  Tag GRX_HomeOk (Scope=)
    PVI Parametreler_0.GRX_HomeOk (Path=Parametreler_0.GRX_HomeOk, Type=Pvar, AccessType=DATA)
      ObjectDescriptor (VT=boolean, VN=1, VL=1, CD=Parametreler_0.GRX_HomeOk, AT=rw, RF=1000, DV=, WR=true)
      LinkDescriptor (BitNumber=none, LT=raw)
        CastMode (Pg2000=false, Decimal=false, Range=false, Rounding=false, TerminateStrings=false)
  Tag GRX_JogNeg (Scope=)
    PVI Parametreler_0.GRX_JogNeg (Path=Parametreler_0.GRX_JogNeg, Type=Pvar, AccessType=DATA)
      ObjectDescriptor (VT=boolean, VN=1, VL=1, CD=Parametreler_0.GRX_JogNeg, AT=rw, RF=1000, DV=, WR=true)
      LinkDescriptor (BitNumber=none, LT=raw)
        CastMode (Pg2000=false, Decimal=false, Range=false, Rounding=false, TerminateStrings=false)
  Tag GRX_JogPos (Scope=)
    PVI Parametreler_0.GRX_JogPos (Path=Parametreler_0.GRX_JogPos, Type=Pvar, AccessType=DATA)
      ObjectDescriptor (VT=boolean, VN=1, VL=1, CD=Parametreler_0.GRX_JogPos, AT=rw, RF=1000, DV=, WR=true)
      LinkDescriptor (BitNumber=none, LT=raw)
        CastMode (Pg2000=false, Decimal=false, Range=false, Rounding=false, TerminateStrings=false)
  Tag GRX_Start_Home (Scope=)
    PVI Parametreler_0.GRX_HomeStart (Path=Parametreler_0.GRX_HomeStart, Type=Pvar, AccessType=DATA)
      ObjectDescriptor (VT=boolean, VN=1, VL=1, CD=Parametreler_0.GRX_HomeStart, AT=rw, RF=1000, DV=, WR=true)
      LinkDescriptor (BitNumber=none, LT=raw)
        CastMode (Pg2000=false, Decimal=false, Range=false, Rounding=false, TerminateStrings=false)
  Tag GRZ_Act_Pos_mm (Scope=)
    PVI Actual_Pos.GRZ_Actual_Pos (Path=Actual_Pos.GRZ_Actual_Pos, Type=Pvar, AccessType=DATA)
      ObjectDescriptor (VT=f32, VN=1, VL=4, CD=Actual_Pos.GRZ_Actual_Pos, AT=rw, RF=1000, DV=, WR=true)
      LinkDescriptor (BitNumber=none, LT=raw)
        CastMode (Pg2000=false, Decimal=false, Range=false, Rounding=false, TerminateStrings=false)
  Tag GRZ_HomeOk (Scope=)
    PVI Parametreler_0.GRZ_HomeOk (Path=Parametreler_0.GRZ_HomeOk, Type=Pvar, AccessType=DATA)
      ObjectDescriptor (VT=boolean, VN=1, VL=1, CD=Parametreler_0.GRZ_HomeOk, AT=rw, RF=1000, DV=, WR=true)
      LinkDescriptor (BitNumber=none, LT=raw)
        CastMode (Pg2000=false, Decimal=false, Range=false, Rounding=false, TerminateStrings=false)
  Tag GRZ_JogNeg (Scope=)
    PVI Parametreler_0.GRZ_JogNeg (Path=Parametreler_0.GRZ_JogNeg, Type=Pvar, AccessType=DATA)
      ObjectDescriptor (VT=boolean, VN=1, VL=1, CD=Parametreler_0.GRZ_JogNeg, AT=rw, RF=1000, DV=, WR=true)
      LinkDescriptor (BitNumber=none, LT=raw)
        CastMode (Pg2000=false, Decimal=false, Range=false, Rounding=false, TerminateStrings=false)
  Tag GRZ_JogPos (Scope=)
    PVI Parametreler_0.GRZ_JogPos (Path=Parametreler_0.GRZ_JogPos, Type=Pvar, AccessType=DATA)
      ObjectDescriptor (VT=boolean, VN=1, VL=1, CD=Parametreler_0.GRZ_JogPos, AT=rw, RF=1000, DV=, WR=true)
      LinkDescriptor (BitNumber=none, LT=raw)
        CastMode (Pg2000=false, Decimal=false, Range=false, Rounding=false, TerminateStrings=false)
  Tag GRZ_Start_Home (Scope=)
    PVI Parametreler_0.GRZ_HomeStart (Path=Parametreler_0.GRZ_HomeStart, Type=Pvar, AccessType=DATA)
      ObjectDescriptor (VT=boolean, VN=1, VL=1, CD=Parametreler_0.GRZ_HomeStart, AT=rw, RF=1000, DV=, WR=true)
      LinkDescriptor (BitNumber=none, LT=raw)
        CastMode (Pg2000=false, Decimal=false, Range=false, Rounding=false, TerminateStrings=false)
  Tag Hatch_Adedi (Scope=)
    PVI Retain.Hatch_Adedi (Path=Retain.Hatch_Adedi, Type=Pvar, AccessType=DATA)
      ObjectDescriptor (VT=i16, VN=1, VL=2, CD=Retain.Hatch_Adedi, AT=rw, RF=1000, DV=, WR=true)
      LinkDescriptor (BitNumber=none, LT=raw)
        CastMode (Pg2000=false, Decimal=false, Range=false, Rounding=false, TerminateStrings=false)
  Tag Krank_Al (Scope=)
    PVI Parametreler_0.Krank_Al (Path=Parametreler_0.Krank_Al, Type=Pvar, AccessType=DATA)
      ObjectDescriptor (VT=boolean, VN=1, VL=1, CD=Parametreler_0.Krank_Al, AT=rw, RF=1000, DV=, WR=true)
      LinkDescriptor (BitNumber=none, LT=raw)
        CastMode (Pg2000=false, Decimal=false, Range=false, Rounding=false, TerminateStrings=false)
  Tag Lazer_Start (Scope=)
    PVI Parametreler_0.Lazer_Start (Path=Parametreler_0.Lazer_Start, Type=Pvar, AccessType=DATA)
      ObjectDescriptor (VT=boolean, VN=1, VL=1, CD=Parametreler_0.Lazer_Start, AT=rw, RF=1000, DV=, WR=true)
      LinkDescriptor (BitNumber=none, LT=raw)
        CastMode (Pg2000=false, Decimal=false, Range=false, Rounding=false, TerminateStrings=false)
  Tag Lazer_Stop (Scope=)
    PVI Parametreler_0.Lazer_Stop (Path=Parametreler_0.Lazer_Stop, Type=Pvar, AccessType=DATA)
      ObjectDescriptor (VT=boolean, VN=1, VL=1, CD=Parametreler_0.Lazer_Stop, AT=rw, RF=1000, DV=, WR=true)
      LinkDescriptor (BitNumber=none, LT=raw)
        CastMode (Pg2000=false, Decimal=false, Range=false, Rounding=false, TerminateStrings=false)
  Tag X_Act_Pos_mm (Scope=)
    PVI Actual_Pos.RX_Actual_Pos (Path=Actual_Pos.RX_Actual_Pos, Type=Pvar, AccessType=DATA)
      ObjectDescriptor (VT=f32, VN=1, VL=4, CD=Actual_Pos.RX_Actual_Pos, AT=rw, RF=1000, DV=, WR=true)
      LinkDescriptor (BitNumber=none, LT=raw)
        CastMode (Pg2000=false, Decimal=false, Range=false, Rounding=false, TerminateStrings=false)
  Tag X_HomeOk (Scope=)
    PVI Parametreler_0.X_HomeOk (Path=Parametreler_0.X_HomeOk, Type=Pvar, AccessType=DATA)
      ObjectDescriptor (VT=boolean, VN=1, VL=1, CD=Parametreler_0.X_HomeOk, AT=rw, RF=1000, DV=, WR=true)
      LinkDescriptor (BitNumber=none, LT=raw)
        CastMode (Pg2000=false, Decimal=false, Range=false, Rounding=false, TerminateStrings=false)
  Tag X_JogNeg (Scope=)
    PVI Parametreler_0.X_JogNeg (Path=Parametreler_0.X_JogNeg, Type=Pvar, AccessType=DATA)
      ObjectDescriptor (VT=boolean, VN=1, VL=1, CD=Parametreler_0.X_JogNeg, AT=rw, RF=1000, DV=, WR=true)
      LinkDescriptor (BitNumber=none, LT=raw)
        CastMode (Pg2000=false, Decimal=false, Range=false, Rounding=false, TerminateStrings=false)
  Tag X_JogPos (Scope=)
    PVI Parametreler_0.X_JogPos (Path=Parametreler_0.X_JogPos, Type=Pvar, AccessType=DATA)
      ObjectDescriptor (VT=boolean, VN=1, VL=1, CD=Parametreler_0.X_JogPos, AT=rw, RF=1000, DV=, WR=true)
      LinkDescriptor (BitNumber=none, LT=raw)
        CastMode (Pg2000=false, Decimal=false, Range=false, Rounding=false, TerminateStrings=false)
  Tag X_Markalama_Konumu (Scope=)
    PVI Retain.RX_MarkalamaKonumu (Path=Retain.RX_MarkalamaKonumu, Type=Pvar, AccessType=DATA)
      ObjectDescriptor (VT=f32, VN=1, VL=4, CD=Retain.RX_MarkalamaKonumu, AT=rw, RF=1000, DV=, WR=true)
      LinkDescriptor (BitNumber=none, LT=raw)
        CastMode (Pg2000=false, Decimal=false, Range=false, Rounding=false, TerminateStrings=false)
  Tag X_Start_Home (Scope=)
    PVI Parametreler_0.X_HomeStart (Path=Parametreler_0.X_HomeStart, Type=Pvar, AccessType=DATA)
      ObjectDescriptor (VT=boolean, VN=1, VL=1, CD=Parametreler_0.X_HomeStart, AT=rw, RF=1000, DV=, WR=true)
      LinkDescriptor (BitNumber=none, LT=raw)
        CastMode (Pg2000=false, Decimal=false, Range=false, Rounding=false, TerminateStrings=false)
  Tag Y_Act_Pos_mm (Scope=)
    PVI Actual_Pos.RY_Actual_Pos (Path=Actual_Pos.RY_Actual_Pos, Type=Pvar, AccessType=DATA)
      ObjectDescriptor (VT=f32, VN=1, VL=4, CD=Actual_Pos.RY_Actual_Pos, AT=rw, RF=1000, DV=, WR=true)
      LinkDescriptor (BitNumber=none, LT=raw)
        CastMode (Pg2000=false, Decimal=false, Range=false, Rounding=false, TerminateStrings=false)
  Tag Y_HomeOk (Scope=)
    PVI Parametreler_0.Y_HomeOk (Path=Parametreler_0.Y_HomeOk, Type=Pvar, AccessType=DATA)
      ObjectDescriptor (VT=boolean, VN=1, VL=1, CD=Parametreler_0.Y_HomeOk, AT=rw, RF=1000, DV=, WR=true)
      LinkDescriptor (BitNumber=none, LT=raw)
        CastMode (Pg2000=false, Decimal=false, Range=false, Rounding=false, TerminateStrings=false)
  Tag Y_JogNeg (Scope=)
    PVI Parametreler_0.Y_JogNeg (Path=Parametreler_0.Y_JogNeg, Type=Pvar, AccessType=DATA)
      ObjectDescriptor (VT=boolean, VN=1, VL=1, CD=Parametreler_0.Y_JogNeg, AT=rw, RF=1000, DV=, WR=true)
      LinkDescriptor (BitNumber=none, LT=raw)
        CastMode (Pg2000=false, Decimal=false, Range=false, Rounding=false, TerminateStrings=false)
  Tag Y_JogPos (Scope=)
    PVI Parametreler_0.Y_JogPos (Path=Parametreler_0.Y_JogPos, Type=Pvar, AccessType=DATA)
      ObjectDescriptor (VT=boolean, VN=1, VL=1, CD=Parametreler_0.Y_JogPos, AT=rw, RF=1000, DV=, WR=true)
      LinkDescriptor (BitNumber=none, LT=raw)
        CastMode (Pg2000=false, Decimal=false, Range=false, Rounding=false, TerminateStrings=false)
  Tag Y_Markalama_Konumu (Scope=)
    PVI Retain.RY_MarkalamaKonumu (Path=Retain.RY_MarkalamaKonumu, Type=Pvar, AccessType=DATA)
      ObjectDescriptor (VT=f32, VN=1, VL=4, CD=Retain.RY_MarkalamaKonumu, AT=rw, RF=1000, DV=, WR=true)
      LinkDescriptor (BitNumber=none, LT=raw)
        CastMode (Pg2000=false, Decimal=false, Range=false, Rounding=false, TerminateStrings=false)
  Tag Y_Start_Home (Scope=)
    PVI Parametreler_0.Y_HomeStart (Path=Parametreler_0.Y_HomeStart, Type=Pvar, AccessType=DATA)
      ObjectDescriptor (VT=boolean, VN=1, VL=1, CD=Parametreler_0.Y_HomeStart, AT=rw, RF=1000, DV=, WR=true)
      LinkDescriptor (BitNumber=none, LT=raw)
        CastMode (Pg2000=false, Decimal=false, Range=false, Rounding=false, TerminateStrings=false)
  Tag Z_Act_Pos_mm (Scope=)
    PVI Actual_Pos.RZ_Actual_Pos (Path=Actual_Pos.RZ_Actual_Pos, Type=Pvar, AccessType=DATA)
      ObjectDescriptor (VT=f32, VN=1, VL=4, CD=Actual_Pos.RZ_Actual_Pos, AT=rw, RF=1000, DV=, WR=true)
      LinkDescriptor (BitNumber=none, LT=raw)
        CastMode (Pg2000=false, Decimal=false, Range=false, Rounding=false, TerminateStrings=false)
  Tag Z_HomeOk (Scope=)
    PVI Parametreler_0.Z_HomeOk (Path=Parametreler_0.Z_HomeOk, Type=Pvar, AccessType=DATA)
      ObjectDescriptor (VT=boolean, VN=1, VL=1, CD=Parametreler_0.Z_HomeOk, AT=rw, RF=1000, DV=, WR=true)
      LinkDescriptor (BitNumber=none, LT=raw)
        CastMode (Pg2000=false, Decimal=false, Range=false, Rounding=false, TerminateStrings=false)
  Tag Z_JogNeg (Scope=)
    PVI Parametreler_0.Z_JogNeg (Path=Parametreler_0.Z_JogNeg, Type=Pvar, AccessType=DATA)
      ObjectDescriptor (VT=boolean, VN=1, VL=1, CD=Parametreler_0.Z_JogNeg, AT=rw, RF=1000, DV=, WR=true)
      LinkDescriptor (BitNumber=none, LT=raw)
        CastMode (Pg2000=false, Decimal=false, Range=false, Rounding=false, TerminateStrings=false)
  Tag Z_JogPos (Scope=)
    PVI Parametreler_0.Z_JogPos (Path=Parametreler_0.Z_JogPos, Type=Pvar, AccessType=DATA)
      ObjectDescriptor (VT=boolean, VN=1, VL=1, CD=Parametreler_0.Z_JogPos, AT=rw, RF=1000, DV=, WR=true)
      LinkDescriptor (BitNumber=none, LT=raw)
        CastMode (Pg2000=false, Decimal=false, Range=false, Rounding=false, TerminateStrings=false)
  Tag Z_Markalama_Konumu (Scope=)
    PVI Retain.RZ_MarkalamaKonumu (Path=Retain.RZ_MarkalamaKonumu, Type=Pvar, AccessType=DATA)
      ObjectDescriptor (VT=f32, VN=1, VL=4, CD=Retain.RZ_MarkalamaKonumu, AT=rw, RF=1000, DV=, WR=true)
      LinkDescriptor (BitNumber=none, LT=raw)
        CastMode (Pg2000=false, Decimal=false, Range=false, Rounding=false, TerminateStrings=false)
  Tag Z_Start_Home (Scope=)
    PVI Parametreler_0.Z_HomeStart (Path=Parametreler_0.Z_HomeStart, Type=Pvar, AccessType=DATA)
      ObjectDescriptor (VT=boolean, VN=1, VL=1, CD=Parametreler_0.Z_HomeStart, AT=rw, RF=1000, DV=, WR=true)
      LinkDescriptor (BitNumber=none, LT=raw)
        CastMode (Pg2000=false, Decimal=false, Range=false, Rounding=false, TerminateStrings=false)
```

### Acp10cfg.ncc - PLC1/Motion/Acp10cfg.ncc
```
NcConfiguration (Version=2.40.1, NcSwId=acp10)
  ACP10CF1_typ:
    cnt_nettrc_rec_drive = 1500
    bufsize_trace_upload = 1200
    tc_nc_man_task = Cyclic #1
    glob_pv_as_ncobject = Yes
    ncsys_dl_broadcast = Yes
    ncsys_dl_acp_reset = Yes
    safemc_log_err_to_ax = Yes
    network_init:
      ncsw_init_execute = Yes
      automatic_execute = No
      node_nr_warning = Yes
      net_err_before_ncact = Yes
    nettrc:
      enter_parsecrec = Yes
      enter_ncaction = Yes
      save_ring_startidx = Yes
    plk_if[0]:
      if_name = SL1.IF1
      tc_CycDat_PLCopen = Task class for NC Manager task
      mc_broadcast_extdat = No
```

### Acp10map.ncm - PLC1/Motion/Acp10map.ncm
```
NcMapping (NcSwId=acp10)
  NcObject gAxis03 (ModuleAddress=SDC_IF1.ST1, InterfaceType=SDC, Type=ncAXIS, Channel=1, AcoposSimulation=Off, InitParameter=x64axisi, AcoposParameter=x64axisa, Disabled=TRUE, ModuleDisabled=FALSE)
  NcObject GX1_Axis (ModuleAddress=SL1.IF1.ST6, InterfaceType=Powerlink, Type=ncAXIS, Channel=1, AcoposSimulation=Off, InitParameter=gaxis02i, AcoposParameter=gaxis02a, Disabled=FALSE, ModuleDisabled=FALSE)
  NcObject SL1.IF1.ST6.VAxis1 (ModuleAddress=SL1.IF1.ST6, InterfaceType=Powerlink, Type=ncV_AXIS, Channel=1, Disabled=TRUE, ModuleDisabled=FALSE)
  NcObject GX2_Axis (ModuleAddress=SL1.IF1.ST6, InterfaceType=Powerlink, Type=ncAXIS, Channel=2, AcoposSimulation=Off, InitParameter=gaxis03i, AcoposParameter=gaxis03a, Disabled=FALSE, ModuleDisabled=FALSE)
  NcObject SL1.IF1.ST6.VAxis2 (ModuleAddress=SL1.IF1.ST6, InterfaceType=Powerlink, Type=ncV_AXIS, Channel=2, Disabled=TRUE, ModuleDisabled=FALSE)
  NcObject GZ1_Axis (ModuleAddress=SL1.IF1.ST7, InterfaceType=Powerlink, Type=ncAXIS, Channel=1, AcoposSimulation=Off, InitParameter=gz1_axisi, AcoposParameter=gz1_axisa, Disabled=FALSE, ModuleDisabled=FALSE)
  NcObject SL1.IF1.ST7.VAxis1 (ModuleAddress=SL1.IF1.ST7, InterfaceType=Powerlink, Type=ncV_AXIS, Channel=1, Disabled=TRUE, ModuleDisabled=FALSE)
  NcObject GC1_Axis (ModuleAddress=SL1.IF1.ST8, InterfaceType=Powerlink, Type=ncAXIS, Channel=1, AcoposSimulation=Off, InitParameter=gc1_axisi, AcoposParameter=gz1_axisa, Disabled=FALSE, ModuleDisabled=FALSE)
  NcObject SL1.IF1.ST8.VAxis1 (ModuleAddress=SL1.IF1.ST8, InterfaceType=Powerlink, Type=ncV_AXIS, Channel=1, Disabled=TRUE, ModuleDisabled=FALSE)
  NcObject GC2_Axis (ModuleAddress=SL1.IF1.ST9, InterfaceType=Powerlink, Type=ncAXIS, Channel=1, AcoposSimulation=Off, InitParameter=gc2_axisi, AcoposParameter=gc2_axisa, Disabled=FALSE, ModuleDisabled=FALSE)
  NcObject GX3_Axis (ModuleAddress=SL1.IF1.ST5, InterfaceType=Powerlink, Type=ncAXIS, Channel=1, AcoposSimulation=Off, InitParameter=gaxis01i, AcoposParameter=gaxis01a, Disabled=FALSE, ModuleDisabled=FALSE)
  NcObject SL1.IF1.ST5.VAxis1 (ModuleAddress=SL1.IF1.ST5, InterfaceType=Powerlink, Type=ncV_AXIS, Channel=1, Disabled=TRUE, ModuleDisabled=FALSE)
  NcObject GRY_Axis (ModuleAddress=SL1.IF1.ST5, InterfaceType=Powerlink, Type=ncAXIS, Channel=2, AcoposSimulation=Off, InitParameter=gry_axisi, AcoposParameter=gry_axisa, Disabled=FALSE, ModuleDisabled=FALSE)
  NcObject SL1.IF1.ST5.VAxis2 (ModuleAddress=SL1.IF1.ST5, InterfaceType=Powerlink, Type=ncV_AXIS, Channel=2, Disabled=TRUE, ModuleDisabled=FALSE)
  NcObject SL1.IF1.ST9.VAxis1 (ModuleAddress=SL1.IF1.ST9, InterfaceType=Powerlink, Type=ncV_AXIS, Channel=1, Disabled=TRUE, ModuleDisabled=FALSE)
  NcObject PowerSp1 (ModuleAddress=SL1.IF1.ST10, InterfaceType=Powerlink, Type=ncAXIS, Channel=1, AcoposSimulation=Off, InitParameter=powersp1i, AcoposParameter=powersp1a, Disabled=FALSE, ModuleDisabled=FALSE)
  NcObject SL1.IF1.ST10.VAxis1 (ModuleAddress=SL1.IF1.ST10, InterfaceType=Powerlink, Type=ncV_AXIS, Channel=1, Disabled=TRUE, ModuleDisabled=FALSE)
  NcObject PowerSp2 (ModuleAddress=SL1.IF1.ST10, InterfaceType=Powerlink, Type=ncAXIS, Channel=2, AcoposSimulation=Off, InitParameter=powersp2i, AcoposParameter=powersp2a, Disabled=FALSE, ModuleDisabled=FALSE)
  NcObject SL1.IF1.ST10.VAxis2 (ModuleAddress=SL1.IF1.ST10, InterfaceType=Powerlink, Type=ncV_AXIS, Channel=2, Disabled=TRUE, ModuleDisabled=FALSE)
  NcObject GRZ_Axis (ModuleAddress=SL1.IF1.ST11, InterfaceType=Powerlink, Type=ncAXIS, Channel=1, AcoposSimulation=Off, InitParameter=grz_axisi, AcoposParameter=grz_axisa, Disabled=FALSE, ModuleDisabled=FALSE)
  NcObject SL1.IF1.ST11.VAxis1 (ModuleAddress=SL1.IF1.ST11, InterfaceType=Powerlink, Type=ncV_AXIS, Channel=1, Disabled=TRUE, ModuleDisabled=FALSE)
  NcObject GRX_Axis (ModuleAddress=SL1.IF1.ST11, InterfaceType=Powerlink, Type=ncAXIS, Channel=2, AcoposSimulation=Off, InitParameter=grx_axisi, AcoposParameter=grx_axisa, Disabled=FALSE, ModuleDisabled=FALSE)
  NcObject SL1.IF1.ST11.VAxis2 (ModuleAddress=SL1.IF1.ST11, InterfaceType=Powerlink, Type=ncV_AXIS, Channel=2, Disabled=TRUE, ModuleDisabled=FALSE)
```

## Logical view

Binary libraries used (declarations not repeated): Operator, runtime, AsTime, AsIecCon, Acp10_MC 2.40.1, brsystem, Acp10man 2.40.1, sys_lib, NcGlobal 2.40.1, Acp10par 2.40.1, Acp10sdc 2.40.1, standard, asstring, AsWeigh, AsBrMath, LoopConR 2.80.9, AsBrStr, FileIO, AsEPL, AsARCfg, dvframe

### Global.typ - Global data types
```iecst
(********************************************************************
 * COPYRIGHT --
 ********************************************************************
 * File: Global.typ
 * Author: Coder
 * Created: September 22, 2013
 ********************************************************************
 * Global data types of project ASILAPC910
 ********************************************************************)

TYPE
	EksenHizlari_typ : 	STRUCT
		X_JogVelocity : REAL;
		Y_JogVelocity : REAL;
		Z_JogVelocity : REAL;
		A_JogVelocity : REAL;
		GRX_JogVelocity : REAL;
		GRY_JogVelocity : REAL;
		GRZ_JogVelocity : REAL;
		GC1_JogVelocity : REAL;
		X_PosVelocity : REAL;
		Y_PosVelocity : REAL;
		Z_PosVelocity : REAL;
		A_PosVelocity : REAL;
		GRX_PosVelocity : REAL;
		GRY_PosVelocity : REAL;
		GRZ_PosVelocity : REAL;
		GC1_PosVelocity : REAL;
	END_STRUCT;
	actual_pos_typ : 	STRUCT
		RX_Actual_Pos : REAL;
		RY_Actual_Pos : REAL;
		RZ_Actual_Pos : REAL;
		RA_Actual_Pos : REAL;
		GRX_Actual_Pos : REAL;
		GRZ_Actual_Pos : REAL;
		GC1_Actual_Pos : REAL;
		GC2_Actual_Pos : REAL;
		GRY_Actual_Pos : REAL;
	END_STRUCT;
	retain_typ : 	STRUCT
		RX_MarkalamaKonumu : REAL;
		RY_MarkalamaKonumu : REAL;
		RZ_MarkalamaKonumu : REAL;
		GRX_KrankKoymaKonumu : REAL;
		GRZ_KrankKoymaKonumu : REAL;
		GRX_KrankAlmaKonumu : REAL;
		GRZ_KrankAlmaKonumu : REAL;
		RA_MarkalamaKonumu : REAL;
		Hatch_Adedi : INT;
		GRX_KrankAlma_Konumu_2 : REAL;
		GRZ_KrankAlma_Konumu_2 : REAL;
		GRX_KrankKoyma_Konumu_2 : REAL;
		GRZ_KrankKoyma_Konumu_2 : REAL;
		Yatay_Sira_Miktari : USINT;
		Dikey_Sira_Miktari : USINT;
		Yatay_Sira_Araligi : REAL;
		Dikey_Sira_Araligi : REAL;
		GRY_KrankAlma_Konumu : REAL;
		GRX_Position : REAL;
		GRZ_Position : REAL;
	END_STRUCT;
	automat_axisState_typ : 	STRUCT  (*axis state structure*)
		Disabled : BOOL; (*if set, axis is in state Disabled*)
		StandStill : BOOL; (*if set, axis is in state StandsStill*)
		Homing : BOOL; (*if set, axis is in state Homing*)
		Stopping : BOOL; (*if set, axis is in state Stopping*)
		DiscreteMotion : BOOL; (*if set, axis is in state DiscreteMotion*)
		ContinuousMotion : BOOL; (*if set, axis is in state ContinuousMotion*)
		SynchronizedMotion : BOOL; (*if set, axis is in state SynchronizedMotion*)
		ErrorStop : BOOL; (*if set, axis is in state ErrorStop*)
	END_STRUCT;
	automat_command_typ : 	STRUCT  (*command structure*)
		Power : BOOL; (*switch on the controller*)
		Home : BOOL; (*reference the axis*)
		MoveAbsolute : BOOL; (*move to an defined position*)
		MoveAdditive : BOOL; (*move a defiened distance*)
		MoveVelocity : BOOL; (*start a movement with a defiened velocity*)
		Halt : BOOL; (*stop every active movement*)
		Stop : BOOL; (*stop every active movement as long as is set*)
		MoveJogPos : BOOL; (*move in positive direction as long as is set*)
		MoveJogNeg : BOOL; (*move in negative direction as long as is set*)
		StartSlave : BOOL; (*start coupling beetween master and slave*)
		StopSlave : BOOL; (*stop coupling between master and slave*)
		GearInPos : BOOL;
		GearOut : BOOL;
		ErrorAcknowledge : BOOL; (*reset active errors*)
	END_STRUCT;
	automat_parameter_typ : 	STRUCT  (*parameter structure*)
		Position : REAL; (*target-position for MoveAbsolute-Command*)
		Distance : REAL; (*distance for MoveAdditive-Command*)
		Velocity : REAL; (*velocity for MoveVelocity-Command*)
		Direction : USINT; (*direction for commanded movements*)
		Acceleration : REAL; (*acceleration for commanded movements*)
		Deceleration : REAL; (*deceleration for commanded movements*)
		HomePosition : REAL; (*target-position for referencing the axis*)
		HomeMode : USINT; (*homing mode*)
		JogVelocity : REAL; (*velocity for jogging movement*)
	END_STRUCT;
	automat_status_typ : 	STRUCT  (*status structure*)
		ErrorID : UINT; (*ErrorID of any occured error*)
		ErrorText : ARRAY[0..3]OF STRING[79]; (*Error Text*)
		ActPosition : REAL; (*actual position of the axis*)
		ActVelocity : REAL; (*actual velocity of the axis*)
		DriveStatus : MC_DRIVESTATUS_TYP; (*actual status of the axis*)
	END_STRUCT;
	automat_typ : 	STRUCT  (*control structure*)
		Command : automat_command_typ; (*command structure*)
		Parameter : automat_parameter_typ; (*parameter structure*)
		Status : automat_status_typ; (*status structure*)
		AxisState : automat_axisState_typ; (*axis state structure*)
		Speed : axis_speed_typ;
	END_STRUCT;
	axis_speed_typ : 	STRUCT
		Manual_Speed : REAL;
		Acceleration : REAL;
		Deceleration : REAL;
		Automatic_Speed : REAL;
		AccelerationOverride : REAL;
		VelocityOverride : REAL;
	END_STRUCT;
	basic_axisState_typ : 	STRUCT  (*axis state structure*)
		Disabled : BOOL; (*if set, axis is in state Disabled*)
		StandStill : BOOL; (*if set, axis is in state StandsStill*)
		Homing : BOOL; (*if set, axis is in state Homing*)
		Stopping : BOOL; (*if set, axis is in state Stopping*)
		DiscreteMotion : BOOL; (*if set, axis is in state DiscreteMotion*)
		ContinuousMotion : BOOL; (*if set, axis is in state ContinuousMotion*)
		SynchronizedMotion : BOOL; (*if set, axis is in state SynchronizedMotion*)
		ErrorStop : BOOL; (*if set, axis is in state ErrorStop*)
	END_STRUCT;
	basic_command_typ : 	STRUCT  (*command structure*)
		Power : BOOL; (*switch on the controller*)
		Home : BOOL; (*reference the axis*)
		MoveAbsolute : BOOL; (*move to an defined position*)
		MoveAdditive : BOOL; (*move a defiened distance*)
		MoveVelocity : BOOL; (*start a movement with a defiened velocity*)
		Halt : BOOL; (*stop every active movement once*)
		Stop : BOOL; (*stop every active movement as long as set*)
		MoveJogPos : BOOL; (*move in positive direction as long as is set*)
		MoveJogNeg : BOOL; (*move in negative direction as long as is set*)
		ErrorAcknowledge : BOOL; (*reset active errors*)
	END_STRUCT;
	basic_parameter_typ : 	STRUCT  (*parameter structure*)
		Position : REAL; (*target-position for MoveAbsolute-Command*)
		Distance : REAL; (*distance for MoveAdditive-Command*)
		Velocity : REAL; (*velocity for MoveVelocity-Command*)
		Direction : USINT; (*direction for commanded movements*)
		Acceleration : REAL; (*acceleration for commanded movements*)
		Deceleration : REAL; (*deceleration for commanded movements*)
		HomePosition : REAL; (*target-position for referencing the axis*)
		HomeMode : USINT; (*homing mode*)
		JogVelocity : REAL; (*velocity for jogging movement*)
	END_STRUCT;
	basic_status_typ : 	STRUCT  (*status structure*)
		ErrorID : UINT; (*ErrorID of any occured error*)
		ErrorText : ARRAY[0..3]OF STRING[79]; (*Error Text*)
		ActPosition : REAL; (*actual position of the axis*)
		ActVelocity : REAL; (*actual velocity of the axis*)
		DriveStatus : MC_DRIVESTATUS_TYP; (*actual status of the axis*)
	END_STRUCT;
	basic_typ : 	STRUCT  (*control structure*)
		Command : basic_command_typ; (*command structure*)
		Parameter : basic_parameter_typ; (*parameter structure*)
		Status : basic_status_typ; (*status structure*)
		AxisState : basic_axisState_typ; (*axis state structure*)
		Speed : axis_speed_typ;
	END_STRUCT;
	Config_setup_typ : 	STRUCT
		LanguageIndex : USINT;
		SubnetMask : ARRAY[0..3]OF USINT;
		IPAddress : ARRAY[0..3]OF USINT;
		Broadcast : ARRAY[0..3]OF USINT;
		Gateway : ARRAY[0..3]OF USINT;
		CmdWriteFile : BOOL;
	END_STRUCT;
	DateTimeStructure_typ : 	STRUCT
		year : UINT;
		month : USINT;
		day : USINT;
		wday : USINT;
		hour : USINT;
		minute : USINT;
		second : USINT;
		millisec : UINT;
		microsec : UINT;
	END_STRUCT;
	digitalinput_typ : 	STRUCT
		Acil_Stop : BOOL;
		X_PosLimit : BOOL;
		X_NegLimit : BOOL;
		X_RefSensor : BOOL;
		Y_NegLimit : BOOL;
		Y_PosLimit : BOOL;
		Y_RefSensor : BOOL;
		Lazer_IsBitti : BOOL;
		GRX_NegLimit : BOOL;
		GRX_RefSensor : BOOL;
		GRX_PosLimit : BOOL;
		GRZ_RefSensor : BOOL;
		GRZ_NegLimit : BOOL;
		GRZ_PosLimit : BOOL;
		GC1_NegLimit : BOOL;
		GC1_RefSensor : BOOL;
		GC1_PosLimit : BOOL;
		GC2_NegLimit : BOOL;
		GC2_RefSensor : BOOL;
		GC2_PosLimit : BOOL;
		GRY_NegLimit : BOOL;
		GRY_PosLimit : BOOL;
		RAnahtarKonumu1 : BOOL;
		RAnahtarKonumu2 : BOOL;
		RAnahtarKonumu3 : BOOL;
		RAnahtarKonumu4 : BOOL;
		R_JoySag : BOOL;
		R_JoySol : BOOL;
		R_Input1 : BOOL;
		LAnahtarKonumu1 : BOOL;
		LAnahtarKonumu2 : BOOL;
		LAnahtarKonumu3 : BOOL;
		LAnahtarKonumu4 : BOOL;
		L_JoySag : BOOL;
		L_JoySol : BOOL;
		L_Input1 : BOOL;
	END_STRUCT;
	digitaloutput_typ : 	STRUCT
		Lazer_Start : BOOL;
		Lazer_Stop : BOOL;
		Lazer_Pointer : BOOL;
		Lazer_Hatch : BOOL;
		Lazer_Barcode : BOOL;
		Konveyor_Ileri : BOOL;
		Konveyor_Geri : BOOL;
		Kripper_Ac : BOOL;
		Kripper_Kapat : BOOL;
	END_STRUCT;
	hmi_ipconfig : 	STRUCT
		EthernetDevice : STRING[10];
		OptionVolatile : UDINT;
		TcpIpReady : USINT;
		IPAddress : ARRAY[0..3]OF USINT;
		SubnetMask : ARRAY[0..3]OF USINT;
		Broadcast : ARRAY[0..3]OF USINT;
		Gateway : ARRAY[0..3]OF USINT;
		EthernetBaudrate : USINT;
		AddressChanged : USINT;
		ReadTcpIp : USINT;
		UpdateTcpIp : USINT;
		ErrorDuringOperation : UINT;
		NodeNumber : USINT;
		cmdLanguageUp : BOOL;
		cmdLanguageDown : BOOL;
		LanguageIndex : USINT;
		LockLanguageUpButton : USINT;
		ActualDateTime : DateTimeStructure_typ;
		DateTimeChanged : USINT;
	END_STRUCT;
	parametreler_typ : 	STRUCT
		X_JogPos : BOOL;
		X_JogNeg : BOOL;
		Y_JogPos : BOOL;
		Y_JogNeg : BOOL;
		Z_JogPos : BOOL;
		Z_JogNeg : BOOL;
		A_JogPos : BOOL;
		A_JogNeg : BOOL;
		X_HomeStart : BOOL;
		Y_HomeStart : BOOL;
		A_HomeStart : BOOL;
		Z_HomeStart : BOOL;
		Alarm_Reset : BOOL;
		Lazer_Start : BOOL;
		Lazer_Stop : BOOL;
		Markalamaya_Git : BOOL;
		X_HomeOk : BOOL;
		Y_HomeOk : BOOL;
		Z_HomeOk : BOOL;
		A_HomeOk : BOOL;
		GRX_JogPos : BOOL;
		GRX_JogNeg : BOOL;
		GRX_HomeStart : BOOL;
		GRX_HomeOk : BOOL;
		GRZ_JogPos : BOOL;
		GRZ_JogNeg : BOOL;
		GRZ_HomeStart : BOOL;
		GRZ_HomeOk : BOOL;
		GC1_HomeStart : BOOL;
		GC1_HomeOk : BOOL;
		GC2_JogPos : BOOL;
		GC2_JogNeg : BOOL;
		GC2_HomeStart : BOOL;
		GC2_HomeOk : BOOL;
		GC1_JogPos : BOOL;
		GC1_JogNeg : BOOL;
		Krank_Al : BOOL;
		Krank_Koy : BOOL;
		Konveyor_Ileri_Buton : BOOL;
		Konveyor_Geri_Buton : BOOL;
		Markalama_Ok : BOOL;
		GRY_HomeStart : BOOL;
		GRY_HomeOk : BOOL;
		GRY_JogNeg : BOOL;
		GRY_JogPos : BOOL;
		Markalama_Start : BOOL;
		Kripper_Ac : BOOL;
		Kripper_Kapat : BOOL;
		Markalama_Ok_Delphi : BOOL;
	END_STRUCT;
	time_typ : 	STRUCT
		XStationLeft : ARRAY[0..9]OF REAL;
		XStationFree : ARRAY[0..9]OF REAL;
		ZStationUp : ARRAY[0..9]OF REAL;
		ZStationDown : ARRAY[0..9]OF REAL;
		Time : ARRAY[0..9]OF UINT;
		TimeUp : ARRAY[0..9]OF UINT;
	END_STRUCT;
END_TYPE
```

### Global.var - Global variables
```iecst
(********************************************************************
 * COPYRIGHT --
 ********************************************************************
 * File: Global.var
 * Author: Coder
 * Created: September 22, 2013
 ********************************************************************
 * Global variables of project ASILAPC910
 ********************************************************************)
VAR RETAIN
	Eksen_Hizlari : EksenHizlari_typ;
END_VAR
VAR
	Actual_Pos : actual_pos_typ;
END_VAR
VAR RETAIN
	Retain : retain_typ;
	admin_password : UDINT;
END_VAR
VAR
	admin_status_group : UINT;
	admin_status_group2 : UINT;
	alarmbits : ARRAY[0..63] OF BOOL;
	DI : digitalinput_typ;
	DQ : digitaloutput_typ;
	GX1_Axis : ACP10AXIS_typ;
	GX1Axis : automat_typ;
	GX2_Axis : ACP10AXIS_typ;
	GX2Axis : automat_typ;
	GX3_Axis : ACP10AXIS_typ;
	GX3Axis : automat_typ;
	GZ1_Axis : ACP10AXIS_typ;
	GZ1Axis : automat_typ;
	GC1_Axis : ACP10AXIS_typ;
	GC1Axis : automat_typ;
	GC2_Axis : ACP10AXIS_typ;
	GC2Axis : automat_typ;
	GRX_Axis : ACP10AXIS_typ;
	GRXAxis : automat_typ;
	GRZ_Axis : ACP10AXIS_typ;
	GRZAxis : automat_typ;
	GRYAxis : automat_typ;
	GRY_Axis : ACP10AXIS_typ;
	PowerSp1 : ACP10AXIS_typ;
	Power1Axis : automat_typ;
	PowerSp2 : ACP10AXIS_typ;
	Power2Axis : automat_typ;
END_VAR
VAR RETAIN
	operator_password : UDINT;
	Parametreler_0 : parametreler_typ;
END_VAR
VAR
	prgname : STRING[9];
	programname : STRING[9];
	Screen : USINT;
END_VAR
VAR RETAIN
	service_password : UDINT;
END_VAR
VAR
	Passwordler : STRING[0];
END_VAR
VAR RETAIN
	Sifre_Ayarlar : UDINT;
END_VAR
VAR
	user_message : STRING[40];
	Sifre_Ayarlar_Giris : BOOL;
	Sifre_Error : BOOL;
END_VAR
VAR RETAIN
	Sifre_Sistem : UDINT;
END_VAR
VAR
	Sifre_Sistem_Giris : BOOL;
END_VAR
VAR RETAIN
	Sifre_Temp_Screen : UDINT;
END_VAR
VAR
	Sifre_Temp : UDINT;
	GX1HomeOk : BOOL;
	GX2HomeOk : BOOL;
	GX3HomeOk : BOOL;
	GZ1HomeOk : BOOL;
	GC2HomeOk : BOOL;
	GC1HomeOk : BOOL;
	GRZHomeOk : BOOL;
	GRXHomeOk : BOOL;
END_VAR
```


### Data object Logical/RYAxisobj/gaxis01i (Ax)

#### gaxis01i.ax
```
InitParameter (Version=2.40.1, NcSwId=acp10)
  ACP10AXIS_typ:
    dig_in:
      level:
        reference = ncACTIV_HI
        pos_hw_end = ncACTIV_HI
        neg_hw_end = ncACTIV_HI
        trigger1 = ncACTIV_HI
        trigger2 = ncACTIV_LO
    encoder_if:
      parameter:
        count_dir = ncSTANDARD
        scaling:
          load:
            units = 1000
            rev_motor = 1
    limit:
      parameter:
        v_pos = 10000
        v_neg = 10000
        a1_pos = 50000
        a2_pos = 50000
        a1_neg = 50000
        a2_neg = 50000
        t_jolt = 0
        t_in_pos = 0
        pos_sw_end = 2000000000
        neg_sw_end = -2000000000
        ds_warning = 500
        ds_stop = 1000
        a_stop = 1.0e30
        dv_stop = 0
        dv_stop_mode = ncOFF
    controller:
      mode = ncPOSITION
      position:
        kv = 50
        tn = 0
        t_predict = 0.0004
        t_total = 0.0004
        p_max = 10000
        i_max = 0
      speed:
        kv = 2.0
        tn = 0
        t_filter = 0.0
        isq_filter1:
          type = ncOFF
          a0 = 0.0
          a1 = 0.0
          b0 = 0.0
          b1 = 0.0
          b2 = 0.0
          c0_par_id = 0
          c1_par_id = 0
        isq_filter2:
          type = ncOFF
          a0 = 0.0
          a1 = 0.0
          b0 = 0.0
          b1 = 0.0
          b2 = 0.0
          c0_par_id = 0
          c1_par_id = 0
        isq_filter3:
          type = ncOFF
          a0 = 0.0
          a1 = 0.0
          b0 = 0.0
          b1 = 0.0
          b2 = 0.0
          c0_par_id = 0
          c1_par_id = 0
      uf:
        type = ncLINEAR
        auto_config = ncMOTOR_PAR
        u0 = 0
        un = 0
        fn = 50.0
        k_f_slip = 0
      ff:
        torque_load = 0.0
        torque_pos = 0.0
        torque_neg = 0.0
        kv_torque = 0.0
        inertia = 0.0
        t_filter_a = 0.0
    move:
      stop:
        parameter[0]:
          decel_ramp = ncA_LIMIT
          controller = ncON
        parameter[1]:
          decel_ramp = ncA_LIMIT
          controller = ncON
        parameter[2]:
          decel_ramp = ncA_LIMIT
          controller = ncON
        parameter[3]:
          decel_ramp = ncA_LIMIT
          controller = ncON
        quickstop:
          decel_ramp = ncA_LIMIT
        drive_error:
          decel_ramp = ncA_LIMIT
      homing:
        parameter:
          s = 0
          v_switch = 5000
          v_trigger = 500
          a = 50000
          mode = ncDIRECT
          edge_sw = ncPOSITIVE
          start_dir = ncPOSITIVE
          trigg_dir = ncPOSITIVE
          ref_pulse = ncOFF
          fix_dir = ncOFF
          tr_s_block = 0
          torque_lim = 0
          ds_block = 0
          ds_stop = 0
      basis:
        parameter:
          v_pos = 5000
          v_neg = 5000
          a1_pos = 50000
          a2_pos = 50000
          a1_neg = 50000
          a2_neg = 50000
    message:
      text:
        parameter:
          format = ncBREAK
          columns = 80
          data_modul = acp10etxen
```

- Data object Logical/RYAxisobj/gaxis01a (Apt) (no source held here)

### Data object Logical/RZAxisobj/gz1_axisi (Ax)

#### gz1_axisi.ax
```
InitParameter (Version=2.40.1, NcSwId=acp10)
  ACP10AXIS_typ:
    dig_in:
      level:
        reference = ncACTIV_HI
        pos_hw_end = ncACTIV_HI
        neg_hw_end = ncACTIV_HI
        trigger1 = ncACTIV_HI
        trigger2 = ncACTIV_LO
    encoder_if:
      parameter:
        count_dir = ncINVERSE
        scaling:
          load:
            units = 1000
            rev_motor = 1
    limit:
      parameter:
        v_pos = 10000
        v_neg = 10000
        a1_pos = 50000
        a2_pos = 50000
        a1_neg = 50000
        a2_neg = 50000
        t_jolt = 0
        t_in_pos = 0
        pos_sw_end = 2000000000
        neg_sw_end = -2000000000
        ds_warning = 500
        ds_stop = 1000
        a_stop = 1.0e30
        dv_stop = 0
        dv_stop_mode = ncOFF
    controller:
      mode = ncPOSITION
      position:
        kv = 50
        tn = 0
        t_predict = 0.0004
        t_total = 0.0004
        p_max = 10000
        i_max = 0
      speed:
        kv = 2.0
        tn = 0
        t_filter = 0.0
        isq_filter1:
          type = ncOFF
          a0 = 0.0
          a1 = 0.0
          b0 = 0.0
          b1 = 0.0
          b2 = 0.0
          c0_par_id = 0
          c1_par_id = 0
        isq_filter2:
          type = ncOFF
          a0 = 0.0
          a1 = 0.0
          b0 = 0.0
          b1 = 0.0
          b2 = 0.0
          c0_par_id = 0
          c1_par_id = 0
        isq_filter3:
          type = ncOFF
          a0 = 0.0
          a1 = 0.0
          b0 = 0.0
          b1 = 0.0
          b2 = 0.0
          c0_par_id = 0
          c1_par_id = 0
      uf:
        type = ncLINEAR
        auto_config = ncMOTOR_PAR
        u0 = 0
        un = 0
        fn = 50.0
        k_f_slip = 0
      ff:
        torque_load = 0.0
        torque_pos = 0.0
        torque_neg = 0.0
        kv_torque = 0.0
        inertia = 0.0
        t_filter_a = 0.0
    move:
      stop:
        parameter[0]:
          decel_ramp = ncA_LIMIT
          controller = ncON
        parameter[1]:
          decel_ramp = ncA_LIMIT
          controller = ncON
        parameter[2]:
          decel_ramp = ncA_LIMIT
          controller = ncON
        parameter[3]:
          decel_ramp = ncA_LIMIT
          controller = ncON
        quickstop:
          decel_ramp = ncA_LIMIT
        drive_error:
          decel_ramp = ncA_LIMIT
      homing:
        parameter:
          s = 0
          v_switch = 5000
          v_trigger = 500
          a = 50000
          mode = ncSWITCH_GATE
          edge_sw = ncPOSITIVE
          start_dir = ncPOSITIVE
          trigg_dir = ncNEGATIVE
          ref_pulse = ncOFF
          fix_dir = ncOFF
          tr_s_block = 0
          torque_lim = 0
          ds_block = 0
          ds_stop = 0
      basis:
        parameter:
          v_pos = 5000
          v_neg = 5000
          a1_pos = 50000
          a2_pos = 50000
          a1_neg = 50000
          a2_neg = 50000
    message:
      text:
        parameter:
          format = ncBREAK
          columns = 80
          data_modul = acp10etxen
```

### Data object Logical/RAAxisobj/gaxis02i (Ax)

#### gaxis02i.ax
```
InitParameter (Version=2.40.1, NcSwId=ACP10)
  ACP10AXIS_typ:
    dig_in:
      level:
        reference = ncACTIV_HI
        pos_hw_end = ncACTIV_LO
        neg_hw_end = ncACTIV_LO
        trigger1 = ncACTIV_HI
        trigger2 = ncACTIV_LO
    encoder_if:
      parameter:
        count_dir = ncSTANDARD
        scaling:
          load:
            units = 1000
            rev_motor = 1
    limit:
      parameter:
        v_pos = 10000
        v_neg = 10000
        a1_pos = 50000
        a2_pos = 50000
        a1_neg = 50000
        a2_neg = 50000
        t_jolt = 0
        t_in_pos = 0
        pos_sw_end = 8388607
        neg_sw_end = -8388608
        ds_warning = 2000.0
        ds_stop = 4000.0
        a_stop = 1e+030
        dv_stop = 0
        dv_stop_mode = ncOFF
    controller:
      mode = ncPOSITION
      position:
        kv = 50
        tn = 0
        t_predict = 0.0004
        t_total = 0.0004
        p_max = 10000
        i_max = 0
      speed:
        kv = 2
        tn = 0
        t_filter = 0
        isq_filter1:
          type = ncOFF
          a0 = 0
          a1 = 0
          b0 = 0
          b1 = 0
          b2 = 0
          c0_par_id = 0
          c1_par_id = 0
        isq_filter2:
          type = ncOFF
          a0 = 0
          a1 = 0
          b0 = 0
          b1 = 0
          b2 = 0
          c0_par_id = 0
          c1_par_id = 0
        isq_filter3:
          type = ncOFF
          a0 = 0
          a1 = 0
          b0 = 0
          b1 = 0
          b2 = 0
          c0_par_id = 0
          c1_par_id = 0
      uf:
        type = ncLINEAR
        auto_config = ncMOTOR_PAR
        u0 = 0
        un = 0
        fn = 50
        k_f_slip = 0
      ff:
        torque_load = 0
        torque_pos = 0
        torque_neg = 0
        kv_torque = 0
        inertia = 0
        t_filter_a = 0
    move:
      stop:
        parameter[0]:
          decel_ramp = ncA_LIMIT
          controller = ncON
        parameter[1]:
          decel_ramp = ncA_LIMIT
          controller = ncON
        parameter[2]:
          decel_ramp = ncA_LIMIT
          controller = ncON
        parameter[3]:
          decel_ramp = ncA_LIMIT
          controller = ncON
        quickstop:
          decel_ramp = ncA_LIMIT
        drive_error:
          decel_ramp = ncA_LIMIT
      homing:
        parameter:
          s = 0
          v_switch = 5000
          v_trigger = 500
          a = 50000
          mode = ncDIRECT
          edge_sw = ncPOSITIVE
          start_dir = ncPOSITIVE
          trigg_dir = ncPOSITIVE
          ref_pulse = ncOFF
          fix_dir = ncOFF
          tr_s_block = 0
          torque_lim = 0
          ds_block = 0
          ds_stop = 0
      basis:
        parameter:
          v_pos = 5000
          v_neg = 5000
          a1_pos = 50000
          a2_pos = 50000
          a1_neg = 50000
          a2_neg = 50000
    message:
      text:
        parameter:
          format = ncBREAK
          columns = 80
          data_modul = acp10etxen
```

### Data object Logical/RAAxisobj/gaxis02a (Apt)

#### gaxis02a.apt
```
AcoposParameterTable:
  Root Parameters:
    390 = 80 (Name=UDC_NOMINAL, Unit=V)  // CTRL DC bus: Nominal voltage
```

### Data object Logical/RXAxisobj/gaxis03i (Ax)

#### gaxis03i.ax
```
InitParameter (Version=2.40.1, NcSwId=ACP10)
  ACP10AXIS_typ:
    dig_in:
      level:
        reference = ncACTIV_HI
        pos_hw_end = ncACTIV_LO
        neg_hw_end = ncACTIV_LO
        trigger1 = ncACTIV_HI
        trigger2 = ncACTIV_LO
    encoder_if:
      parameter:
        count_dir = ncSTANDARD
        scaling:
          load:
            units = 1000
            rev_motor = 1
    limit:
      parameter:
        v_pos = 10000
        v_neg = 10000
        a1_pos = 50000
        a2_pos = 50000
        a1_neg = 50000
        a2_neg = 50000
        t_jolt = 0
        t_in_pos = 0
        pos_sw_end = 8388607
        neg_sw_end = -39140
        ds_warning = 500
        ds_stop = 1000
        a_stop = 1e+030
        dv_stop = 0
        dv_stop_mode = ncOFF
    controller:
      mode = ncPOSITION
      position:
        kv = 50
        tn = 0
        t_predict = 0.0004
        t_total = 0.0004
        p_max = 10000
        i_max = 0
      speed:
        kv = 2
        tn = 0
        t_filter = 0
        isq_filter1:
          type = ncOFF
          a0 = 0
          a1 = 0
          b0 = 0
          b1 = 0
          b2 = 0
          c0_par_id = 0
          c1_par_id = 0
        isq_filter2:
          type = ncOFF
          a0 = 0
          a1 = 0
          b0 = 0
          b1 = 0
          b2 = 0
          c0_par_id = 0
          c1_par_id = 0
        isq_filter3:
          type = ncOFF
          a0 = 0
          a1 = 0
          b0 = 0
          b1 = 0
          b2 = 0
          c0_par_id = 0
          c1_par_id = 0
      uf:
        type = ncLINEAR
        auto_config = ncMOTOR_PAR
        u0 = 0
        un = 0
        fn = 50
        k_f_slip = 0
      ff:
        torque_load = 0
        torque_pos = 0
        torque_neg = 0
        kv_torque = 0
        inertia = 0
        t_filter_a = 0
    move:
      stop:
        parameter[0]:
          decel_ramp = ncA_LIMIT
          controller = ncON
        parameter[1]:
          decel_ramp = ncA_LIMIT
          controller = ncON
        parameter[2]:
          decel_ramp = ncA_LIMIT
          controller = ncON
        parameter[3]:
          decel_ramp = ncA_LIMIT
          controller = ncON
        quickstop:
          decel_ramp = ncA_LIMIT
        drive_error:
          decel_ramp = ncA_LIMIT
      homing:
        parameter:
          s = 0
          v_switch = 5000
          v_trigger = 500
          a = 50000
          mode = ncDIRECT
          edge_sw = ncPOSITIVE
          start_dir = ncPOSITIVE
          trigg_dir = ncPOSITIVE
          ref_pulse = ncOFF
          fix_dir = ncOFF
          tr_s_block = 0
          torque_lim = 0
          ds_block = 0
          ds_stop = 0
      basis:
        parameter:
          v_pos = 5000
          v_neg = 5000
          a1_pos = 50000
          a2_pos = 50000
          a1_neg = 50000
          a2_neg = 50000
    message:
      text:
        parameter:
          format = ncBREAK
          columns = 80
          data_modul = acp10etxen
```

### Data object Logical/RXAxisobj/gaxis03a (Apt)

#### gaxis03a.apt
```
AcoposParameterTable:
  Root Parameters:
    390 = 80 (Name=UDC_NOMINAL, Unit=V)  // CTRL DC bus: Nominal voltage
```

### Data object Logical/RC1Axisobj/gc1_axisi (Ax)

#### gz1_axisi.ax
```
InitParameter (Version=2.40.1, NcSwId=acp10)
  ACP10AXIS_typ:
    dig_in:
      level:
        reference = ncACTIV_HI
        pos_hw_end = ncACTIV_HI
        neg_hw_end = ncACTIV_HI
        trigger1 = ncACTIV_HI
        trigger2 = ncACTIV_LO
    encoder_if:
      parameter:
        count_dir = ncSTANDARD
        scaling:
          load:
            units = 1000
            rev_motor = 1
    limit:
      parameter:
        v_pos = 10000
        v_neg = 10000
        a1_pos = 50000
        a2_pos = 50000
        a1_neg = 50000
        a2_neg = 50000
        t_jolt = 0
        t_in_pos = 0
        pos_sw_end = 29700
        neg_sw_end = -200
        ds_warning = 500
        ds_stop = 10000.0
        a_stop = 1.0e30
        dv_stop = 0
        dv_stop_mode = ncOFF
    controller:
      mode = ncPOSITION
      position:
        kv = 200.0
        tn = 0
        t_predict = 0.0004
        t_total = 0.0004
        p_max = 10000
        i_max = 0
      speed:
        kv = 4.0
        tn = 0
        t_filter = 0.0008
        isq_filter1:
          type = ncOFF
          a0 = 0.0
          a1 = 0.0
          b0 = 0.0
          b1 = 0.0
          b2 = 0.0
          c0_par_id = 0
          c1_par_id = 0
        isq_filter2:
          type = ncOFF
          a0 = 0.0
          a1 = 0.0
          b0 = 0.0
          b1 = 0.0
          b2 = 0.0
          c0_par_id = 0
          c1_par_id = 0
        isq_filter3:
          type = ncOFF
          a0 = 0.0
          a1 = 0.0
          b0 = 0.0
          b1 = 0.0
          b2 = 0.0
          c0_par_id = 0
          c1_par_id = 0
      uf:
        type = ncLINEAR
        auto_config = ncMOTOR_PAR
        u0 = 0
        un = 0
        fn = 50.0
        k_f_slip = 0
      ff:
        torque_load = 0.0
        torque_pos = 0.0
        torque_neg = 0.0
        kv_torque = 0.0
        inertia = 0.0
        t_filter_a = 0.0
    move:
      stop:
        parameter[0]:
          decel_ramp = ncA_LIMIT
          controller = ncON
        parameter[1]:
          decel_ramp = ncA_LIMIT
          controller = ncON
        parameter[2]:
          decel_ramp = ncA_LIMIT
          controller = ncON
        parameter[3]:
          decel_ramp = ncA_LIMIT
          controller = ncON
        quickstop:
          decel_ramp = ncA_LIMIT
        drive_error:
          decel_ramp = ncA_LIMIT
      homing:
        parameter:
          s = 0
          v_switch = 500.0
          v_trigger = 200.0
          a = 50000
          mode = ncSWITCH_GATE
          edge_sw = ncNEGATIVE
          start_dir = ncNEGATIVE
          trigg_dir = ncPOSITIVE
          ref_pulse = ncOFF
          fix_dir = ncOFF
          tr_s_block = 0
          torque_lim = 0
          ds_block = 0
          ds_stop = 0
      basis:
        parameter:
          v_pos = 5000
          v_neg = 5000
          a1_pos = 50000
          a2_pos = 50000
          a1_neg = 50000
          a2_neg = 50000
    message:
      text:
        parameter:
          format = ncBREAK
          columns = 80
          data_modul = acp10etxen
```

### Data object Logical/RC2Axisobj/gc2_axisi (Ax)

#### gz1_axisi.ax
```
InitParameter (Version=2.40.1, NcSwId=acp10)
  ACP10AXIS_typ:
    dig_in:
      level:
        reference = ncACTIV_HI
        pos_hw_end = ncACTIV_HI
        neg_hw_end = ncACTIV_HI
        trigger1 = ncACTIV_HI
        trigger2 = ncACTIV_LO
    encoder_if:
      parameter:
        count_dir = ncINVERSE
        scaling:
          load:
            units = 1000
            rev_motor = 1
    limit:
      parameter:
        v_pos = 10000
        v_neg = 10000
        a1_pos = 50000
        a2_pos = 50000
        a1_neg = 50000
        a2_neg = 50000
        t_jolt = 0
        t_in_pos = 0
        pos_sw_end = 29700
        neg_sw_end = -200
        ds_warning = 500
        ds_stop = 10000.0
        a_stop = 1.0e30
        dv_stop = 0
        dv_stop_mode = ncOFF
    controller:
      mode = ncPOSITION
      position:
        kv = 200.0
        tn = 0
        t_predict = 0.0004
        t_total = 0.0004
        p_max = 10000
        i_max = 0
      speed:
        kv = 4.0
        tn = 0
        t_filter = 0.0008
        isq_filter1:
          type = ncOFF
          a0 = 0.0
          a1 = 0.0
          b0 = 0.0
          b1 = 0.0
          b2 = 0.0
          c0_par_id = 0
          c1_par_id = 0
        isq_filter2:
          type = ncOFF
          a0 = 0.0
          a1 = 0.0
          b0 = 0.0
          b1 = 0.0
          b2 = 0.0
          c0_par_id = 0
          c1_par_id = 0
        isq_filter3:
          type = ncOFF
          a0 = 0.0
          a1 = 0.0
          b0 = 0.0
          b1 = 0.0
          b2 = 0.0
          c0_par_id = 0
          c1_par_id = 0
      uf:
        type = ncLINEAR
        auto_config = ncMOTOR_PAR
        u0 = 0
        un = 0
        fn = 50.0
        k_f_slip = 0
      ff:
        torque_load = 0.0
        torque_pos = 0.0
        torque_neg = 0.0
        kv_torque = 0.0
        inertia = 0.0
        t_filter_a = 0.0
    move:
      stop:
        parameter[0]:
          decel_ramp = ncA_LIMIT
          controller = ncON
        parameter[1]:
          decel_ramp = ncA_LIMIT
          controller = ncON
        parameter[2]:
          decel_ramp = ncA_LIMIT
          controller = ncON
        parameter[3]:
          decel_ramp = ncA_LIMIT
          controller = ncON
        quickstop:
          decel_ramp = ncA_LIMIT
        drive_error:
          decel_ramp = ncA_LIMIT
      homing:
        parameter:
          s = 0
          v_switch = 500.0
          v_trigger = 200.0
          a = 50000
          mode = ncSWITCH_GATE
          edge_sw = ncNEGATIVE
          start_dir = ncNEGATIVE
          trigg_dir = ncPOSITIVE
          ref_pulse = ncOFF
          fix_dir = ncOFF
          tr_s_block = 0
          torque_lim = 0
          ds_block = 0
          ds_stop = 0
      basis:
        parameter:
          v_pos = 5000
          v_neg = 5000
          a1_pos = 50000
          a2_pos = 50000
          a1_neg = 50000
          a2_neg = 50000
    message:
      text:
        parameter:
          format = ncBREAK
          columns = 80
          data_modul = acp10etxen
```

### Data object Logical/GRXAxisobj/grx_axisi (Ax)

#### gz1_axisi.ax
```
InitParameter (Version=2.40.1, NcSwId=acp10)
  ACP10AXIS_typ:
    dig_in:
      level:
        reference = ncACTIV_HI
        pos_hw_end = ncACTIV_HI
        neg_hw_end = ncACTIV_HI
        trigger1 = ncACTIV_HI
        trigger2 = ncACTIV_LO
    encoder_if:
      parameter:
        count_dir = ncINVERSE
        scaling:
          load:
            units = 1000
            rev_motor = 1
    limit:
      parameter:
        v_pos = 100000.0
        v_neg = 100000.0
        a1_pos = 500000.0
        a2_pos = 500000.0
        a1_neg = 500000.0
        a2_neg = 500000.0
        t_jolt = 0
        t_in_pos = 0
        pos_sw_end = 2000000000
        neg_sw_end = -2000000000
        ds_warning = 500.0
        ds_stop = 5000.0
        a_stop = 1.0e30
        dv_stop = 0
        dv_stop_mode = ncOFF
    controller:
      mode = ncPOSITION
      position:
        kv = 400.0
        tn = 0
        t_predict = 0.0004
        t_total = 0.0004
        p_max = 10000
        i_max = 0
      speed:
        kv = 5.0
        tn = 0
        t_filter = 0.0008
        isq_filter1:
          type = ncOFF
          a0 = 0.0
          a1 = 0.0
          b0 = 0.0
          b1 = 0.0
          b2 = 0.0
          c0_par_id = 0
          c1_par_id = 0
        isq_filter2:
          type = ncOFF
          a0 = 0.0
          a1 = 0.0
          b0 = 0.0
          b1 = 0.0
          b2 = 0.0
          c0_par_id = 0
          c1_par_id = 0
        isq_filter3:
          type = ncOFF
          a0 = 0.0
          a1 = 0.0
          b0 = 0.0
          b1 = 0.0
          b2 = 0.0
          c0_par_id = 0
          c1_par_id = 0
      uf:
        type = ncLINEAR
        auto_config = ncMOTOR_PAR
        u0 = 0
        un = 0
        fn = 50.0
        k_f_slip = 0
      ff:
        torque_load = 0.0
        torque_pos = 0.0
        torque_neg = 0.0
        kv_torque = 0.0
        inertia = 0.0
        t_filter_a = 0.0
    move:
      stop:
        parameter[0]:
          decel_ramp = ncA_LIMIT
          controller = ncON
        parameter[1]:
          decel_ramp = ncA_LIMIT
          controller = ncON
        parameter[2]:
          decel_ramp = ncA_LIMIT
          controller = ncON
        parameter[3]:
          decel_ramp = ncA_LIMIT
          controller = ncON
        quickstop:
          decel_ramp = ncA_LIMIT
        drive_error:
          decel_ramp = ncA_LIMIT
      homing:
        parameter:
          s = 0
          v_switch = 5000.0
          v_trigger = 500.0
          a = 10000.0
          mode = ncDIRECT
          edge_sw = ncPOSITIVE
          start_dir = ncPOSITIVE
          trigg_dir = ncPOSITIVE
          ref_pulse = ncOFF
          fix_dir = ncOFF
          tr_s_block = 0
          torque_lim = 0
          ds_block = 0
          ds_stop = 0
      basis:
        parameter:
          v_pos = 100000.0
          v_neg = 100000.0
          a1_pos = 50000.0
          a2_pos = 50000.0
          a1_neg = 50000.0
          a2_neg = 50000.0
    message:
      text:
        parameter:
          format = ncBREAK
          columns = 80
          data_modul = acp10etxen
```

### Data object Logical/GRXAxisobj/grx_axisa (Apt)

#### gz1_axisa.apt
```
AcoposParameterTable:
  Root Parameters:
    390 = 500 (Name=UDC_NOMINAL, Unit=V)  // CTRL DC bus: Nominal voltage
```

### Package Logical/GRYAxisobj - An empty package

### Data object Logical/GRYAxisobj/gry_axisi (Ax) - ACP10: Axis data object.

#### gry_axisi.ax
```
InitParameter (Version=2.40.1, NcSwId=ACP10)
  ACP10AXIS_typ:
    dig_in:
      level:
        reference = ncACTIV_HI
        pos_hw_end = ncACTIV_HI
        neg_hw_end = ncACTIV_HI
        trigger1 = ncACTIV_HI
        trigger2 = ncACTIV_LO
    encoder_if:
      parameter:
        count_dir = ncSTANDARD
        scaling:
          load:
            units = 1000
            rev_motor = 1
    limit:
      parameter:
        v_pos = 10000
        v_neg = 10000
        a1_pos = 50000
        a2_pos = 50000
        a1_neg = 50000
        a2_neg = 50000
        t_jolt = 0
        t_in_pos = 0
        pos_sw_end = 2000000000
        neg_sw_end = -2000000000
        ds_warning = 500
        ds_stop = 1000
        a_stop = 1.0e30
        dv_stop = 0
        dv_stop_mode = ncOFF
    controller:
      mode = ncPOSITION
      position:
        kv = 50
        tn = 0
        t_predict = 0.0004
        t_total = 0.0004
        p_max = 1.0e30
        i_max = 0
      speed:
        kv = 2.0
        tn = 0
        t_filter = 0.0
        isq_filter1:
          type = ncOFF
          a0 = 0.0
          a1 = 0.0
          b0 = 0.0
          b1 = 0.0
          b2 = 0.0
          c0_par_id = 0
          c1_par_id = 0
        isq_filter2:
          type = ncOFF
          a0 = 0.0
          a1 = 0.0
          b0 = 0.0
          b1 = 0.0
          b2 = 0.0
          c0_par_id = 0
          c1_par_id = 0
        isq_filter3:
          type = ncOFF
          a0 = 0.0
          a1 = 0.0
          b0 = 0.0
          b1 = 0.0
          b2 = 0.0
          c0_par_id = 0
          c1_par_id = 0
      uf:
        type = ncLINEAR
        auto_config = ncMOTOR_PAR
        u0 = 0
        un = 0
        fn = 50.0
        k_f_slip = 0
      ff:
        torque_load = 0.0
        torque_pos = 0.0
        torque_neg = 0.0
        kv_torque = 0.0
        inertia = 0.0
        t_filter_a = 0.0
    move:
      stop:
        parameter[0]:
          decel_ramp = ncA_LIMIT
          controller = ncON
        parameter[1]:
          decel_ramp = ncA_LIMIT
          controller = ncON
        parameter[2]:
          decel_ramp = ncA_LIMIT
          controller = ncON
        parameter[3]:
          decel_ramp = ncA_LIMIT
          controller = ncON
        quickstop:
          decel_ramp = ncA_LIMIT
        drive_error:
          decel_ramp = ncA_LIMIT
      homing:
        parameter:
          s = 0
          v_switch = 5000
          v_trigger = 500
          a = 50000
          mode = ncDIRECT
          edge_sw = ncPOSITIVE
          start_dir = ncPOSITIVE
          trigg_dir = ncPOSITIVE
          ref_pulse = ncOFF
          fix_dir = ncOFF
          tr_s_block = 0
          torque_lim = 0
          ds_block = 0
          ds_stop = 0
      basis:
        parameter:
          v_pos = 5000
          v_neg = 5000
          a1_pos = 50000
          a2_pos = 50000
          a1_neg = 50000
          a2_neg = 50000
    message:
      text:
        parameter:
          format = ncBREAK
          columns = 80
          data_modul
```

- Data object Logical/GRYAxisobj/gry_axisa (Apt) - ACOPOS Parameter Table (no source held here)

### Data object Logical/GRZAxisobj/grz_axisi (Ax)

#### gz1_axisi.ax
```
InitParameter (Version=2.40.1, NcSwId=acp10)
  ACP10AXIS_typ:
    dig_in:
      level:
        reference = ncACTIV_HI
        pos_hw_end = ncACTIV_HI
        neg_hw_end = ncACTIV_HI
        trigger1 = ncACTIV_HI
        trigger2 = ncACTIV_LO
    encoder_if:
      parameter:
        count_dir = ncSTANDARD
        scaling:
          load:
            units = 1000
            rev_motor = 1
    limit:
      parameter:
        v_pos = 100000.0
        v_neg = 100000.0
        a1_pos = 500000.0
        a2_pos = 500000.0
        a1_neg = 500000.0
        a2_neg = 500000.0
        t_jolt = 0
        t_in_pos = 0
        pos_sw_end = 2000000000
        neg_sw_end = -2000000000
        ds_warning = 500
        ds_stop = 1000
        a_stop = 1.0e30
        dv_stop = 0
        dv_stop_mode = ncOFF
    controller:
      mode = ncPOSITION
      position:
        kv = 200.0
        tn = 0
        t_predict = 0.0004
        t_total = 0.0004
        p_max = 10000
        i_max = 0
      speed:
        kv = 4.0
        tn = 0
        t_filter = 0.0008
        isq_filter1:
          type = ncOFF
          a0 = 0.0
          a1 = 0.0
          b0 = 0.0
          b1 = 0.0
          b2 = 0.0
          c0_par_id = 0
          c1_par_id = 0
        isq_filter2:
          type = ncOFF
          a0 = 0.0
          a1 = 0.0
          b0 = 0.0
          b1 = 0.0
          b2 = 0.0
          c0_par_id = 0
          c1_par_id = 0
        isq_filter3:
          type = ncOFF
          a0 = 0.0
          a1 = 0.0
          b0 = 0.0
          b1 = 0.0
          b2 = 0.0
          c0_par_id = 0
          c1_par_id = 0
      uf:
        type = ncLINEAR
        auto_config = ncMOTOR_PAR
        u0 = 0
        un = 0
        fn = 50.0
        k_f_slip = 0
      ff:
        torque_load = 0.0
        torque_pos = 0.0
        torque_neg = 0.0
        kv_torque = 0.0
        inertia = 0.0
        t_filter_a = 0.0
    move:
      stop:
        parameter[0]:
          decel_ramp = ncA_LIMIT
          controller = ncON
        parameter[1]:
          decel_ramp = ncA_LIMIT
          controller = ncON
        parameter[2]:
          decel_ramp = ncA_LIMIT
          controller = ncON
        parameter[3]:
          decel_ramp = ncA_LIMIT
          controller = ncON
        quickstop:
          decel_ramp = ncA_LIMIT
        drive_error:
          decel_ramp = ncA_LIMIT
      homing:
        parameter:
          s = 0
          v_switch = 10000.0
          v_trigger = 500
          a = 50000
          mode = ncDIRECT
          edge_sw = ncPOSITIVE
          start_dir = ncPOSITIVE
          trigg_dir = ncPOSITIVE
          ref_pulse = ncOFF
          fix_dir = ncOFF
          tr_s_block = 0
          torque_lim = 0
          ds_block = 0
          ds_stop = 0
      basis:
        parameter:
          v_pos = 50000.0
          v_neg = 50000.0
          a1_pos = 50000
          a2_pos = 50000
          a1_neg = 50000
          a2_neg = 50000
    message:
      text:
        parameter:
          format = ncBREAK
          columns = 80
          data_modul = acp10etxen
```

- Data object Logical/GRZAxisobj/grz_axisa (Apt) (no source held here)

- Data object Logical/PowerSp1obj/powersp1i (Ax) (no source held here)

### Data object Logical/PowerSp1obj/powersp1a (Apt)

#### powersp1a.apt
```
AcoposParameterTable:
  Root Parameters:
    8B0W0045H000.001-1 mounting vertical V1:
       DO NOT USE with ACOPOS Firmware before V2.27.0 (Disabled=FALSE)
        10 = 50 (Name=R_BLEEDER_EXT, Unit=Ohm, Disabled=FALSE)  // Bleeder: External: Resistance
        11 = 682.65 (Name=TEMP_MAX_BLEEDER_EXT, Unit=°C, Disabled=FALSE)  // Bleeder: External: Limit temperature
        12 = 1.517 (Name=RTH_BLEEDER_AMB_EXT, Unit=K/W, Disabled=FALSE)  // Bleeder: External: Thermal resistance
        13 = 30.88 (Name=CTH_BLEEDER_EXT, Unit=Ws/K, Disabled=FALSE)  // Bleeder: External: Thermal capacity
        398 = 1 (Name=BLEEDER_SELECTOR_EXT, Disabled=FALSE)  // Bleeder: Selector
    390 = 500 (Name=UDC_NOMINAL, Unit=V)  // CTRL DC bus: Nominal voltage
```

### Data object Logical/PowerSp2obj/powersp2i (Ax)
